C08939=1018.974,60.779,-109.447,166.802,53.022,159.705
C08940=1018.980,61.027,-109.462,166.804,53.016,159.704
C08941=1018.986,61.276,-109.479,166.807,53.009,159.704
C08942=1018.991,61.526,-109.494,166.810,53.001,159.703
C08943=1018.997,61.776,-109.511,166.812,52.995,159.702
C08944=1019.002,62.025,-109.526,166.815,52.987,159.701
C08945=1019.007,62.275,-109.543,166.817,52.981,159.700
C08946=1019.013,62.524,-109.559,166.820,52.973,159.700
C08947=1019.019,62.774,-109.574,166.822,52.967,159.699
C08948=1019.025,63.023,-109.591,166.825,52.960,159.698
C08949=1019.030,63.272,-109.607,166.827,52.953,159.697
C08950=1019.036,63.522,-109.623,166.831,52.946,159.697
C08951=1019.042,63.771,-109.640,166.833,52.939,159.696
C08952=1019.046,64.021,-109.656,166.836,52.932,159.695
C08953=1019.052,64.270,-109.672,166.838,52.926,159.694
C08954=1019.057,64.520,-109.688,166.841,52.918,159.693
C08955=1019.063,64.769,-109.705,166.844,52.912,159.693
C08956=1019.069,65.018,-109.721,166.847,52.905,159.692
C08957=1019.074,65.268,-109.738,166.849,52.898,159.691
C08958=1019.079,65.517,-109.754,166.852,52.891,159.690
C08959=1019.084,65.767,-109.770,166.854,52.884,159.689
C08960=1019.090,66.016,-109.786,166.856,52.878,159.688
C08961=1019.096,66.266,-109.803,166.859,52.871,159.688
C08962=1019.101,66.515,-109.819,166.862,52.865,159.687
C08963=1019.106,66.764,-109.836,166.865,52.857,159.686
C08964=1019.112,67.014,-109.852,166.867,52.851,159.685
C08965=1019.118,67.263,-109.868,166.870,52.843,159.684
C08966=1019.123,67.513,-109.885,166.872,52.837,159.684
C08967=1019.129,67.762,-109.901,166.875,52.830,159.683
C08968=1019.134,68.011,-109.918,166.877,52.823,159.682
C08969=1019.140,68.260,-109.934,166.881,52.816,159.681
C08970=1019.145,68.510,-109.951,166.883,52.810,159.680
C08971=1019.150,68.760,-109.968,166.886,52.802,159.680
C08972=1019.156,69.009,-109.984,166.888,52.796,159.679
C08973=1019.161,69.259,-110.001,166.890,52.789,159.678
C08974=1019.167,69.507,-110.017,166.894,52.782,159.677
C08975=1019.172,69.757,-110.034,166.896,52.776,159.676
C08976=1019.177,70.007,-110.050,166.899,52.769,159.676
C08977=1019.183,70.256,-110.067,166.901,52.762,159.675
C08978=1019.188,70.506,-110.084,166.904,52.755,159.674
C08979=1019.194,70.755,-110.100,166.906,52.748,159.673
C08980=1019.199,71.005,-110.117,166.910,52.742,159.673
C08981=1019.204,71.254,-110.133,166.912,52.735,159.672
C08982=1019.210,71.502,-110.150,166.914,52.728,159.671
C08983=1019.216,71.752,-110.167,166.917,52.721,159.670
C08984=1019.221,72.002,-110.184,166.919,52.714,159.669
C08985=1019.227,72.251,-110.200,166.922,52.707,159.668
C08986=1019.232,72.501,-110.217,166.925,52.701,159.668
C08987=1019.238,72.750,-110.233,166.928,52.694,159.667
C08988=1019.243,73.000,-110.250,166.930,52.687,159.666
C08989=1019.248,73.249,-110.267,166.933,52.680,159.665
C08990=1019.254,73.497,-110.284,166.935,52.673,159.664
C08991=1019.259,73.747,-110.300,166.939,52.666,159.664
C08992=1019.264,73.997,-110.317,166.941,52.659,159.663
C08993=1019.270,74.246,-110.333,166.944,52.653,159.662
C08994=1019.276,74.496,-110.350,166.946,52.646,159.661
C08995=1019.282,74.778,-110.369,166.949,52.638,159.660
C08996=1019.288,75.061,-110.389,166.952,52.631,159.659
C08997=1019.294,75.343,-110.408,166.956,52.622,159.658
C08998=1019.300,75.626,-110.427,166.958,52.615,159.657
C08999=1019.306,75.875,-110.443,166.960,52.608,159.657
C09000=1019.311,76.125,-110.460,166.964,52.601,159.656
C09001=1019.317,76.374,-110.477,166.966,52.595,159.655
C09002=1019.322,76.623,-110.494,166.969,52.588,159.654
C09003=1019.328,76.873,-110.510,166.971,52.581,159.653
C09004=1019.333,77.122,-110.528,166.974,52.574,159.653
C09005=1019.339,77.371,-110.545,166.977,52.567,159.652
C09006=1019.344,77.621,-110.562,166.979,52.560,159.651
C09007=1019.349,77.870,-110.579,166.982,52.554,159.650
C09008=1019.355,78.120,-110.596,166.984,52.547,159.649
C09009=1019.360,78.369,-110.613,166.988,52.540,159.649
C09010=1019.365,78.619,-110.630,166.990,52.533,159.648
C09011=1019.371,78.868,-110.647,166.993,52.527,159.647
C09012=1019.376,79.117,-110.665,166.995,52.520,159.646
C09013=1019.381,79.367,-110.682,166.998,52.514,159.645
C09014=1019.388,79.616,-110.699,167.001,52.506,159.645
C09015=1019.393,79.865,-110.716,167.003,52.500,159.644
C09016=1019.398,80.115,-110.732,167.006,52.493,159.643
C09017=1019.403,80.364,-110.750,167.009,52.487,159.642
C09018=1019.408,80.613,-110.766,167.012,52.480,159.642
C09019=1019.414,80.862,-110.784,167.014,52.473,159.641
C09020=1019.419,81.112,-110.801,167.016,52.466,159.640
C09021=1019.424,81.361,-110.818,167.019,52.459,159.639
C09022=1019.430,81.610,-110.835,167.021,52.452,159.638
C09023=1019.436,81.860,-110.853,167.025,52.446,159.638
C09024=1019.441,82.110,-110.870,167.027,52.439,159.637
C09025=1019.446,82.359,-110.888,167.030,52.432,159.636
C09026=1019.452,82.608,-110.905,167.032,52.425,159.635
C09027=1019.457,82.857,-110.922,167.036,52.418,159.634
C09028=1019.462,83.107,-110.939,167.038,52.412,159.633
C09029=1019.468,83.356,-110.956,167.041,52.404,159.633
C09030=1019.473,83.606,-110.973,167.043,52.398,159.632
C09031=1019.479,83.855,-110.991,167.047,52.391,159.631
C09032=1019.485,84.104,-111.007,167.049,52.385,159.630
C09033=1019.490,84.353,-111.025,167.051,52.378,159.629
C09034=1019.495,84.603,-111.042,167.054,52.371,159.629
C09035=1019.501,84.852,-111.059,167.056,52.364,159.628
C09036=1019.506,85.102,-111.076,167.059,52.357,159.627
C09037=1019.512,85.351,-111.094,167.062,52.350,159.626
C09038=1019.517,85.600,-111.111,167.065,52.343,159.625
C09039=1019.522,85.849,-111.128,167.067,52.337,159.624
C09040=1019.528,86.098,-111.146,167.070,52.330,159.624
C09041=1019.533,86.348,-111.162,167.072,52.323,159.623
C09042=1019.539,86.597,-111.180,167.075,52.316,159.622
C09043=1019.545,86.847,-111.198,167.078,52.309,159.621
C09044=1019.550,87.096,-111.215,167.081,52.302,159.620
C09045=1019.555,87.346,-111.232,167.083,52.295,159.619
C09046=1019.561,87.595,-111.249,167.086,52.288,159.619
C09047=1019.566,87.844,-111.267,167.088,52.282,159.618
C09048=1019.572,88.093,-111.284,167.092,52.275,159.617
C09049=1019.577,88.343,-111.301,167.095,52.267,159.616
C09050=1019.582,88.592,-111.319,167.097,52.261,159.615
C09051=1019.588,88.841,-111.336,167.100,52.254,159.615
C09052=1019.594,89.091,-111.354,167.103,52.248,159.614
C09053=1019.599,89.340,-111.371,167.106,52.241,159.613
C09054=1019.605,89.589,-111.389,167.108,52.234,159.612
C09055=1019.610,89.838,-111.406,167.110,52.227,159.611
C09056=1019.615,90.088,-111.424,167.113,52.220,159.611
C09057=1019.620,90.337,-111.441,167.116,52.214,159.610
C09058=1019.626,90.587,-111.459,167.119,52.207,159.609
C09059=1019.632,90.870,-111.479,167.122,52.199,159.608
C09060=1019.638,91.152,-111.500,167.125,52.192,159.607
C09061=1019.644,91.435,-111.519,167.128,52.184,159.606
C09062=1019.650,91.718,-111.539,167.131,52.177,159.605
C09063=1019.655,91.967,-111.557,167.134,52.170,159.605
C09064=1019.661,92.216,-111.574,167.136,52.163,159.604
C09065=1019.666,92.466,-111.593,167.139,52.156,159.603
C09066=1019.672,92.715,-111.610,167.142,52.150,159.602
C09067=1019.677,92.964,-111.628,167.145,52.142,159.601
C09068=1019.682,93.213,-111.646,167.147,52.136,159.601
C09069=1019.687,93.463,-111.663,167.150,52.129,159.600
C09070=1019.693,93.712,-111.680,167.152,52.122,159.599
C09071=1019.699,93.962,-111.698,167.156,52.116,159.598
C09072=1019.704,94.211,-111.716,167.158,52.109,159.597
C09073=1019.709,94.460,-111.734,167.161,52.102,159.597
C09074=1019.715,94.709,-111.752,167.164,52.095,159.596
C09075=1019.720,94.958,-111.769,167.167,52.088,159.595
C09076=1019.726,95.208,-111.788,167.169,52.082,159.594
C09077=1019.731,95.457,-111.805,167.172,52.075,159.593
C09078=1019.737,95.706,-111.823,167.174,52.068,159.592
C09079=1019.742,95.956,-111.841,167.178,52.061,159.592
C09080=1019.747,96.205,-111.859,167.180,52.054,159.591
C09081=1019.753,96.454,-111.876,167.183,52.047,159.590
C09082=1019.759,96.703,-111.894,167.185,52.041,159.589
C09083=1019.763,96.953,-111.912,167.189,52.034,159.588
C09084=1019.769,97.202,-111.930,167.191,52.027,159.587
C09085=1019.775,97.452,-111.948,167.194,52.020,159.587
C09086=1019.781,97.701,-111.965,167.196,52.013,159.586
C09087=1019.785,97.950,-111.983,167.199,52.006,159.585
C09088=1019.791,98.199,-112.001,167.202,52.000,159.584
C09089=1019.797,98.449,-112.019,167.205,51.993,159.583
C09090=1019.802,98.698,-112.037,167.207,51.986,159.583
C09091=1019.807,98.947,-112.055,167.210,51.979,159.582
C09092=1019.813,99.196,-112.072,167.214,51.972,159.581
C09093=1019.818,99.446,-112.091,167.216,51.965,159.580
C09094=1019.824,99.695,-112.108,167.218,51.959,159.579
C09095=1019.829,99.945,-112.126,167.222,51.952,159.579
C09096=1019.835,100.194,-112.144,167.224,51.946,159.578
C09097=1019.840,100.443,-112.163,167.227,51.939,159.577
C09098=1019.845,100.692,-112.181,167.229,51.932,159.576
C09099=1019.850,100.942,-112.199,167.233,51.925,159.575
C09100=1019.855,101.192,-112.218,167.235,51.918,159.574
C09101=1019.861,101.441,-112.235,167.239,51.912,159.574
C09102=1019.866,101.689,-112.254,167.241,51.905,159.573
C09103=1019.872,101.938,-112.272,167.244,51.898,159.572
C09104=1019.877,102.188,-112.290,167.246,51.892,159.571
C09105=1019.882,102.438,-112.308,167.249,51.885,159.571
C09106=1019.888,102.686,-112.327,167.252,51.878,159.570
C09107=1019.893,102.936,-112.345,167.255,51.871,159.569
C09108=1019.898,103.185,-112.363,167.257,51.864,159.568
C09109=1019.903,103.435,-112.381,167.260,51.857,159.567
C09110=1019.910,103.684,-112.399,167.263,51.851,159.567
C09111=1019.914,103.933,-112.418,167.266,51.844,159.566
C09112=1019.919,104.182,-112.436,167.269,51.838,159.565
C09113=1019.925,104.432,-112.454,167.272,51.831,159.564
C09114=1019.930,104.681,-112.473,167.274,51.824,159.563
C09115=1019.936,104.930,-112.490,167.277,51.817,159.563
C09116=1019.941,105.180,-112.509,167.280,51.811,159.562
C09117=1019.946,105.429,-112.528,167.283,51.804,159.561
C09118=1019.952,105.678,-112.545,167.285,51.797,159.560
C09119=1019.957,105.928,-112.564,167.288,51.790,159.559
C09120=1019.963,106.176,-112.582,167.292,51.783,159.559
C09121=1019.968,106.426,-112.600,167.294,51.776,159.558
C09122=1019.974,106.675,-112.618,167.297,51.769,159.557
C09123=1019.979,106.958,-112.640,167.300,51.762,159.556
C09124=1019.986,107.241,-112.660,167.303,51.754,159.555
C09125=1019.992,107.524,-112.681,167.307,51.746,159.554
C09126=1019.998,107.806,-112.702,167.310,51.738,159.553
C09127=1020.004,108.056,-112.720,167.312,51.732,159.552
C09128=1020.009,108.305,-112.738,167.315,51.725,159.551
C09129=1020.014,108.554,-112.757,167.318,51.718,159.551
C09130=1020.020,108.804,-112.775,167.321,51.711,159.550
C09131=1020.025,109.052,-112.794,167.324,51.704,159.549
C09132=1020.032,109.302,-112.812,167.326,51.698,159.548
C09133=1020.036,109.551,-112.830,167.330,51.691,159.547
C09134=1020.041,109.800,-112.849,167.332,51.684,159.546
C09135=1020.047,110.050,-112.867,167.335,51.678,159.546
C09136=1020.053,110.299,-112.885,167.338,51.671,159.545
C09137=1020.058,110.549,-112.904,167.341,51.664,159.544
C09138=1020.063,110.797,-112.923,167.344,51.657,159.543
C09139=1020.068,111.047,-112.941,167.347,51.651,159.543
C09140=1020.074,111.296,-112.960,167.350,51.644,159.542
C09141=1020.079,111.545,-112.979,167.352,51.637,159.541
C09142=1020.085,111.795,-112.997,167.355,51.630,159.540
C09143=1020.090,112.043,-113.016,167.358,51.623,159.539
C09144=1020.095,112.293,-113.034,167.361,51.616,159.539
C09145=1020.100,112.542,-113.053,167.363,51.610,159.538
C09146=1020.106,112.792,-113.073,167.367,51.603,159.537
C09147=1020.111,113.041,-113.091,167.369,51.597,159.536
C09148=1020.116,113.290,-113.110,167.373,51.590,159.535
C09149=1020.122,113.539,-113.129,167.375,51.583,159.535
C09150=1020.127,113.789,-113.147,167.378,51.576,159.534
C09151=1020.132,114.038,-113.166,167.380,51.570,159.533
C09152=1020.137,114.287,-113.185,167.384,51.564,159.532
C09153=1020.143,114.536,-113.204,167.386,51.557,159.531
C09154=1020.148,114.785,-113.223,167.390,51.550,159.531
C09155=1020.153,115.035,-113.242,167.392,51.543,159.530
C09156=1020.158,115.284,-113.261,167.395,51.536,159.529
C09157=1020.164,115.533,-113.280,167.398,51.530,159.528
C09158=1020.169,115.782,-113.298,167.401,51.523,159.527
C09159=1020.175,116.032,-113.317,167.404,51.517,159.527
C09160=1020.179,116.281,-113.337,167.407,51.510,159.526
C09161=1020.185,116.530,-113.356,167.409,51.504,159.525
C09162=1020.190,116.779,-113.375,167.412,51.497,159.524
C09163=1020.195,117.029,-113.393,167.415,51.490,159.523
C09164=1020.200,117.278,-113.412,167.418,51.483,159.523
C09165=1020.206,117.527,-113.432,167.421,51.476,159.522
C09166=1020.211,117.776,-113.450,167.424,51.470,159.521
C09167=1020.217,118.025,-113.470,167.427,51.463,159.520
C09168=1020.222,118.274,-113.489,167.430,51.457,159.520
C09169=1020.227,118.524,-113.507,167.433,51.450,159.519
C09170=1020.232,118.773,-113.526,167.435,51.443,159.518
C09171=1020.238,119.022,-113.545,167.439,51.436,159.517
C09172=1020.243,119.271,-113.564,167.441,51.430,159.516
C09173=1020.249,119.521,-113.583,167.444,51.423,159.516
C09174=1020.254,119.770,-113.603,167.448,51.416,159.515
C09175=1020.259,120.019,-113.622,167.450,51.409,159.514
C09176=1020.264,120.268,-113.641,167.454,51.403,159.513
C09177=1020.269,120.517,-113.660,167.456,51.396,159.512
C09178=1020.275,120.767,-113.679,167.459,51.390,159.512
C09179=1020.280,121.016,-113.698,167.463,51.383,159.511
C09180=1020.286,121.265,-113.717,167.465,51.376,159.510
C09181=1020.291,121.515,-113.736,167.468,51.369,159.509
C09182=1020.296,121.764,-113.755,167.471,51.363,159.508
C09183=1020.302,122.013,-113.774,167.474,51.356,159.508
C09184=1020.307,122.262,-113.793,167.477,51.349,159.507
C09185=1020.313,122.511,-113.812,167.480,51.342,159.506
C09186=1020.318,122.761,-113.832,167.483,51.335,159.505
C09187=1020.324,123.043,-113.853,167.486,51.328,159.504
C09188=1020.330,123.326,-113.875,167.490,51.320,159.503
C09189=1020.336,123.609,-113.897,167.493,51.312,159.502
C09190=1020.342,123.891,-113.918,167.496,51.305,159.502
C09191=1020.348,124.141,-113.938,167.499,51.298,159.501
C09192=1020.353,124.389,-113.957,167.503,51.291,159.500
C09193=1020.359,124.639,-113.976,167.505,51.285,159.499
C09194=1020.364,124.889,-113.996,167.508,51.278,159.498
C09195=1020.369,125.137,-114.015,167.512,51.271,159.498
C09196=1020.375,125.387,-114.034,167.514,51.264,159.497
C09197=1020.380,125.636,-114.053,167.517,51.257,159.496
C09198=1020.385,125.885,-114.072,167.520,51.251,159.495
C09199=1020.391,126.134,-114.091,167.523,51.244,159.494
C09200=1020.397,126.384,-114.110,167.526,51.237,159.494
C09201=1020.402,126.633,-114.129,167.530,51.230,159.493
C09202=1020.408,126.882,-114.148,167.532,51.224,159.492
C09203=1020.413,127.131,-114.168,167.536,51.217,159.491
C09204=1020.418,127.380,-114.188,167.539,51.210,159.490
C09205=1020.424,127.629,-114.207,167.541,51.203,159.489
C09206=1020.429,127.879,-114.226,167.544,51.196,159.489
C09207=1020.435,128.128,-114.246,167.548,51.189,159.488
C09208=1020.440,128.377,-114.265,167.550,51.182,159.487
C09209=1020.446,128.626,-114.284,167.553,51.175,159.486
C09210=1020.451,128.876,-114.303,167.557,51.169,159.485
C09211=1020.456,129.124,-114.322,167.559,51.162,159.484
C09212=1020.462,129.374,-114.341,167.562,51.155,159.484
C09213=1020.468,129.623,-114.361,167.566,51.148,159.483
C09214=1020.473,129.872,-114.381,167.569,51.141,159.482
C09215=1020.478,130.121,-114.400,167.571,51.135,159.481
C09216=1020.484,130.371,-114.419,167.575,51.128,159.481
C09217=1020.489,130.620,-114.440,167.577,51.122,159.480
C09218=1020.495,130.869,-114.459,167.581,51.115,159.479
C09219=1020.500,131.119,-114.479,167.584,51.108,159.478
C09220=1020.505,131.368,-114.498,167.587,51.102,159.477
C09221=1020.510,131.617,-114.518,167.590,51.095,159.477
C09222=1020.516,131.866,-114.537,167.593,51.088,159.476
C09223=1020.520,132.115,-114.558,167.596,51.082,159.475
C09224=1020.526,132.364,-114.577,167.599,51.075,159.474
C09225=1020.532,132.614,-114.596,167.603,51.068,159.474
C09226=1020.537,132.863,-114.617,167.605,51.062,159.473
C09227=1020.543,133.112,-114.636,167.609,51.055,159.472
C09228=1020.547,133.361,-114.655,167.611,51.049,159.471
C09229=1020.553,133.610,-114.675,167.614,51.042,159.470
C09230=1020.558,133.860,-114.695,167.618,51.035,159.470
C09231=1020.564,134.108,-114.715,167.620,51.028,159.469
C09232=1020.568,134.358,-114.735,167.623,51.021,159.468
C09233=1020.574,134.606,-114.754,167.627,51.015,159.467
C09234=1020.579,134.856,-114.774,167.630,51.008,159.466
C09235=1020.585,135.106,-114.794,167.633,51.001,159.466
C09236=1020.591,135.354,-114.814,167.636,50.995,159.465
C09237=1020.595,135.603,-114.833,167.640,50.988,159.464
C09238=1020.601,135.852,-114.853,167.642,50.982,159.463
C09239=1020.606,136.102,-114.873,167.645,50.975,159.463
C09240=1020.612,136.351,-114.893,167.649,50.968,159.462
C09241=1020.617,136.600,-114.913,167.651,50.961,159.461
C09242=1020.623,136.850,-114.933,167.655,50.955,159.460
C09243=1020.628,137.098,-114.952,167.658,50.948,159.459
C09244=1020.633,137.347,-114.973,167.660,50.941,159.459
C09245=1020.639,137.596,-114.993,167.664,50.934,159.458
C09246=1020.644,137.846,-115.012,167.668,50.928,159.457
C09247=1020.650,138.095,-115.032,167.671,50.921,159.456
C09248=1020.655,138.345,-115.052,167.673,50.915,159.456
C09249=1020.659,138.593,-115.072,167.677,50.908,159.455
C09250=1020.665,138.842,-115.092,167.680,50.901,159.454
C09251=1020.671,139.125,-115.115,167.683,50.894,159.453
C09252=1020.677,139.408,-115.138,167.687,50.887,159.452
C09253=1020.684,139.690,-115.161,167.691,50.879,159.451
C09254=1020.689,139.973,-115.184,167.694,50.871,159.450
C09255=1020.695,140.222,-115.204,167.697,50.864,159.450
C09256=1020.700,140.472,-115.224,167.701,50.858,159.449
C09257=1020.705,140.720,-115.244,167.703,50.852,159.448
C09258=1020.710,140.969,-115.264,167.707,50.845,159.447
C09259=1020.716,141.219,-115.284,167.710,50.838,159.447
C09260=1020.721,141.468,-115.304,167.712,50.832,159.446
C09261=1020.726,141.717,-115.325,167.716,50.825,159.445
C09262=1020.732,141.966,-115.345,167.719,50.818,159.444
C09263=1020.737,142.215,-115.365,167.723,50.812,159.444
C09264=1020.743,142.464,-115.385,167.725,50.805,159.443
C09265=1020.748,142.714,-115.406,167.729,50.799,159.442
C09266=1020.754,142.962,-115.426,167.732,50.792,159.441
C09267=1020.759,143.212,-115.445,167.735,50.785,159.440
C09268=1020.763,143.461,-115.466,167.738,50.778,159.440
C09269=1020.769,143.710,-115.486,167.742,50.772,159.439
C09270=1020.775,143.959,-115.506,167.745,50.765,159.438
C09271=1020.780,144.208,-115.527,167.748,50.759,159.437
C09272=1020.785,144.457,-115.547,167.751,50.752,159.437
C09273=1020.790,144.707,-115.567,167.755,50.745,159.436
C09274=1020.796,144.955,-115.587,167.758,50.738,159.435
C09275=1020.801,145.204,-115.608,167.760,50.732,159.434
C09276=1020.807,145.454,-115.628,167.764,50.725,159.433
C09277=1020.813,145.702,-115.648,167.767,50.718,159.433
C09278=1020.818,145.952,-115.669,167.771,50.712,159.432
C09279=1020.823,146.201,-115.689,167.774,50.706,159.431
C09280=1020.828,146.450,-115.710,167.777,50.699,159.430
C09281=1020.834,146.699,-115.730,167.780,50.692,159.430
C09282=1020.839,146.949,-115.750,167.784,50.685,159.429
C09283=1020.844,147.198,-115.771,167.787,50.680,159.428
C09284=1020.849,147.447,-115.791,167.790,50.673,159.427
C09285=1020.854,147.696,-115.812,167.794,50.666,159.427
C09286=1020.860,147.945,-115.832,167.797,50.659,159.426
C09287=1020.865,148.194,-115.854,167.800,50.653,159.425
C09288=1020.870,148.443,-115.874,167.803,50.647,159.424
C09289=1020.876,148.692,-115.895,167.807,50.640,159.424
C09290=1020.881,148.941,-115.915,167.810,50.633,159.423
C09291=1020.886,149.190,-115.936,167.812,50.626,159.422
C09292=1020.891,149.439,-115.956,167.816,50.620,159.421
C09293=1020.897,149.688,-115.977,167.820,50.614,159.421
C09294=1020.902,149.938,-115.998,167.823,50.607,159.420
C09295=1020.907,150.187,-116.018,167.826,50.600,159.419
C09296=1020.912,150.436,-116.039,167.829,50.594,159.418
C09297=1020.918,150.685,-116.059,167.833,50.587,159.418
C09298=1020.923,150.934,-116.080,167.836,50.581,159.417
C09299=1020.929,151.183,-116.101,167.839,50.574,159.416
C09300=1020.934,151.432,-116.122,167.842,50.567,159.415
C09301=1020.940,151.681,-116.142,167.846,50.561,159.415
C09302=1020.945,151.931,-116.163,167.850,50.554,159.414
C09303=1020.950,152.180,-116.184,167.853,50.548,159.413
C09304=1020.955,152.429,-116.204,167.855,50.541,159.412
C09305=1020.961,152.677,-116.225,167.859,50.534,159.411
C09306=1020.966,152.926,-116.246,167.863,50.528,159.411
C09307=1020.971,153.176,-116.267,167.866,50.522,159.410
C09308=1020.977,153.425,-116.287,167.870,50.515,159.409
C09309=1020.982,153.674,-116.308,167.872,50.508,159.408
C09310=1020.988,153.923,-116.329,167.876,50.502,159.408
C09311=1020.993,154.172,-116.350,167.879,50.495,159.407
C09312=1020.999,154.421,-116.370,167.883,50.489,159.406
C09313=1021.003,154.670,-116.392,167.887,50.483,159.406
C09314=1021.009,154.919,-116.413,167.889,50.476,159.405
C09315=1021.015,155.201,-116.437,167.893,50.468,159.404
C09316=1021.021,155.484,-116.460,167.897,50.462,159.403
C09317=1021.027,155.766,-116.484,167.901,50.454,159.402
C09318=1021.033,156.050,-116.507,167.905,50.446,159.402
C09319=1021.039,156.298,-116.529,167.908,50.440,159.401
C09320=1021.043,156.548,-116.550,167.911,50.433,159.400
C09321=1021.049,156.797,-116.570,167.915,50.427,159.399
C09322=1021.054,157.045,-116.592,167.918,50.420,159.399
C09323=1021.059,157.294,-116.612,167.922,50.414,159.398
C09324=1021.066,157.543,-116.634,167.926,50.407,159.397
C09325=1021.071,157.793,-116.654,167.928,50.401,159.396
C09326=1021.075,158.042,-116.676,167.931,50.394,159.396
C09327=1021.081,158.291,-116.697,167.935,50.388,159.395
C09328=1021.086,158.540,-116.717,167.939,50.381,159.394
C09329=1021.092,158.789,-116.739,167.942,50.374,159.393
C09330=1021.098,159.038,-116.760,167.946,50.368,159.393
C09331=1021.102,159.287,-116.781,167.949,50.362,159.392
C09332=1021.107,159.536,-116.803,167.952,50.356,159.391
C09333=1021.113,159.785,-116.824,167.956,50.349,159.391
C09334=1021.117,160.034,-116.846,167.959,50.342,159.390
C09335=1021.123,160.283,-116.868,167.962,50.337,159.389
C09336=1021.128,160.532,-116.888,167.966,50.330,159.388
C09337=1021.133,160.781,-116.910,167.970,50.324,159.388
C09338=1021.138,161.030,-116.932,167.973,50.317,159.387
C09339=1021.143,161.279,-116.953,167.976,50.311,159.386
C09340=1021.148,161.528,-116.975,167.979,50.304,159.386
C09341=1021.154,161.777,-116.996,167.983,50.298,159.385
C09342=1021.159,162.026,-117.018,167.987,50.292,159.384
C09343=1021.163,162.275,-117.039,167.991,50.286,159.384
C09344=1021.169,162.524,-117.061,167.993,50.279,159.383
C09345=1021.174,162.773,-117.083,167.997,50.273,159.382
C09346=1021.180,163.022,-117.104,168.000,50.266,159.381
C09347=1021.184,163.271,-117.125,168.004,50.260,159.381
C09348=1021.189,163.520,-117.147,168.008,50.254,159.380
C09349=1021.195,163.769,-117.169,168.011,50.248,159.379
C09350=1021.200,164.018,-117.191,168.014,50.241,159.379
C09351=1021.205,164.267,-117.212,168.018,50.235,159.378
C09352=1021.211,164.517,-117.233,168.022,50.228,159.377
C09353=1021.216,164.765,-117.255,168.025,50.222,159.377
C09354=1021.221,165.014,-117.277,168.028,50.216,159.376
C09355=1021.226,165.263,-117.298,168.031,50.209,159.375
C09356=1021.231,165.512,-117.321,168.035,50.203,159.374
C09357=1021.237,165.761,-117.342,168.039,50.196,159.374
C09358=1021.242,166.010,-117.363,168.043,50.190,159.373
C09359=1021.247,166.260,-117.385,168.046,50.184,159.372
C09360=1021.253,166.508,-117.406,168.050,50.178,159.372
C09361=1021.257,166.757,-117.428,168.053,50.171,159.371
C09362=1021.263,167.007,-117.451,168.056,50.165,159.370
C09363=1021.268,167.255,-117.472,168.060,50.158,159.370
C09364=1021.273,167.504,-117.494,168.064,50.152,159.369
C09365=1021.279,167.753,-117.516,168.067,50.146,159.368
C09366=1021.284,168.002,-117.537,168.071,50.140,159.368
C09367=1021.289,168.251,-117.559,168.075,50.133,159.367
C09368=1021.294,168.500,-117.581,168.078,50.126,159.366
C09369=1021.300,168.749,-117.603,168.082,50.120,159.365
C09370=1021.305,168.998,-117.624,168.085,50.114,159.365
C09371=1021.311,169.247,-117.645,168.089,50.108,159.364
C09372=1021.315,169.496,-117.667,168.092,50.101,159.363
C09373=1021.321,169.746,-117.689,168.096,50.095,159.363
C09374=1021.326,169.994,-117.711,168.100,50.088,159.362
C09375=1021.331,170.243,-117.733,168.103,50.082,159.361
C09376=1021.337,170.493,-117.755,168.107,50.076,159.360
C09377=1021.342,170.741,-117.776,168.111,50.070,159.360
C09378=1021.348,170.990,-117.799,168.114,50.063,159.359
C09379=1021.354,171.272,-117.823,168.119,50.056,159.358
C09380=1021.360,171.554,-117.849,168.122,50.048,159.357
C09381=1021.366,171.836,-117.873,168.127,50.041,159.357
C09382=1021.372,172.118,-117.898,168.131,50.034,159.356
C09383=1021.377,172.367,-117.920,168.135,50.028,159.355
C09384=1021.383,172.617,-117.942,168.138,50.021,159.355
C09385=1021.388,172.865,-117.963,168.142,50.015,159.354
C09386=1021.394,173.115,-117.985,168.146,50.008,159.353
C09387=1021.398,173.364,-118.007,168.150,50.002,159.353
C09388=1021.405,173.613,-118.029,168.153,49.996,159.352
C09389=1021.409,173.862,-118.051,168.157,49.989,159.351
C09390=1021.415,174.111,-118.074,168.161,49.983,159.350
C09391=1021.421,174.359,-118.095,168.164,49.976,159.350
C09392=1021.426,174.609,-118.117,168.168,49.970,159.349
C09393=1021.431,174.857,-118.139,168.171,49.964,159.348
C09394=1021.437,175.107,-118.161,168.175,49.957,159.348
C09395=1021.442,175.355,-118.183,168.179,49.951,159.347
C09396=1021.448,175.604,-118.205,168.183,49.945,159.346
C09397=1021.453,175.853,-118.227,168.186,49.938,159.346
C09398=1021.459,176.102,-118.249,168.190,49.931,159.345
C09399=1021.464,176.352,-118.271,168.194,49.925,159.344
C09400=1021.470,176.600,-118.293,168.197,49.919,159.343
C09401=1021.475,176.849,-118.315,168.201,49.913,159.343
C09402=1021.480,177.098,-118.337,168.205,49.906,159.342
C09403=1021.486,177.347,-118.359,168.209,49.900,159.341
C09404=1021.492,177.595,-118.381,168.212,49.893,159.341
C09405=1021.497,177.845,-118.404,168.216,49.887,159.340
C09406=1021.502,178.095,-118.426,168.220,49.881,159.339
C09407=1021.508,178.343,-118.447,168.223,49.874,159.339
C09408=1021.514,178.592,-118.470,168.227,49.868,159.338
C09409=1021.518,178.841,-118.492,168.231,49.861,159.337
C09410=1021.525,179.090,-118.514,168.236,49.855,159.337
C09411=1021.530,179.339,-118.537,168.239,49.848,159.336
C09412=1021.535,179.588,-118.558,168.243,49.842,159.335
C09413=1021.541,179.837,-118.580,168.247,49.836,159.335
C09414=1021.547,180.086,-118.603,168.251,49.830,159.334
C09415=1021.552,180.335,-118.625,168.254,49.823,159.333
C09416=1021.558,180.584,-118.647,168.258,49.817,159.333
C09417=1021.564,180.833,-118.669,168.262,49.810,159.332
C09418=1021.569,181.081,-118.691,168.265,49.804,159.331
C09419=1021.575,181.330,-118.714,168.270,49.798,159.331
C09420=1021.581,181.580,-118.736,168.274,49.791,159.330
C09421=1021.586,181.828,-118.759,168.278,49.785,159.329
C09422=1021.591,182.077,-118.781,168.281,49.778,159.328
C09423=1021.597,182.327,-118.803,168.285,49.772,159.328
C09424=1021.602,182.575,-118.826,168.289,49.766,159.327
C09425=1021.607,182.824,-118.848,168.293,49.760,159.326
C09426=1021.612,183.074,-118.871,168.297,49.754,159.326
C09427=1021.618,183.323,-118.894,168.301,49.748,159.325
C09428=1021.623,183.571,-118.917,168.305,49.742,159.325
C09429=1021.628,183.820,-118.940,168.308,49.736,159.324
C09430=1021.633,184.070,-118.963,168.312,49.729,159.323
C09431=1021.638,184.318,-118.985,168.316,49.723,159.323
C09432=1021.644,184.567,-119.008,168.320,49.717,159.322
C09433=1021.649,184.816,-119.032,168.324,49.711,159.322
C09434=1021.654,185.064,-119.054,168.327,49.705,159.321
C09435=1021.660,185.314,-119.076,168.331,49.699,159.320
C09436=1021.665,185.563,-119.100,168.335,49.693,159.320
C09437=1021.670,185.811,-119.123,168.339,49.687,159.319
C09438=1021.676,186.060,-119.146,168.343,49.681,159.318
C09439=1021.681,186.309,-119.169,168.347,49.674,159.318
C09440=1021.686,186.558,-119.192,168.351,49.668,159.317
C09441=1021.691,186.806,-119.215,168.355,49.662,159.316
C09442=1021.696,187.056,-119.237,168.359,49.656,159.316
C09443=1021.702,187.338,-119.264,168.363,49.649,159.315
C09444=1021.708,187.619,-119.290,168.368,49.642,159.314
C09445=1021.714,187.901,-119.316,168.372,49.635,159.314
C09446=1021.720,188.183,-119.342,168.377,49.628,159.313
C09447=1021.726,188.431,-119.364,168.381,49.622,159.312
C09448=1021.731,188.680,-119.387,168.385,49.616,159.312
C09449=1021.736,188.929,-119.411,168.388,49.610,159.311
C09450=1021.742,189.178,-119.434,168.392,49.604,159.310
C09451=1021.748,189.427,-119.457,168.396,49.598,159.310
C09452=1021.752,189.676,-119.480,168.401,49.591,159.309
C09453=1021.758,189.924,-119.503,168.405,49.585,159.309
C09454=1021.764,190.173,-119.526,168.409,49.579,159.308
C09455=1021.769,190.423,-119.549,168.413,49.573,159.307
C09456=1021.774,190.671,-119.572,168.417,49.567,159.307
C09457=1021.780,190.920,-119.595,168.420,49.561,159.306
C09458=1021.784,191.169,-119.619,168.424,49.555,159.305
C09459=1021.790,191.418,-119.641,168.429,49.549,159.305
C09460=1021.796,191.667,-119.664,168.433,49.543,159.304
C09461=1021.801,191.916,-119.688,168.437,49.537,159.304
C09462=1021.807,192.165,-119.711,168.441,49.531,159.303
C09463=1021.813,192.413,-119.735,168.445,49.524,159.302
C09464=1021.818,192.662,-119.758,168.449,49.518,159.302
C09465=1021.823,192.911,-119.781,168.454,49.512,159.301
C09466=1021.828,193.160,-119.804,168.458,49.506,159.301
C09467=1021.834,193.409,-119.827,168.462,49.500,159.300
C09468=1021.839,193.657,-119.850,168.465,49.493,159.299
C09469=1021.844,193.907,-119.874,168.469,49.488,159.299
C09470=1021.850,194.156,-119.897,168.474,49.481,159.298
C09471=1021.856,194.404,-119.920,168.478,49.475,159.298
C09472=1021.861,194.653,-119.944,168.482,49.469,159.297
C09473=1021.867,194.902,-119.967,168.486,49.464,159.296
C09474=1021.872,195.151,-119.990,168.490,49.457,159.296
C09475=1021.877,195.400,-120.013,168.495,49.451,159.295
C09476=1021.883,195.648,-120.037,168.499,49.445,159.295
C09477=1021.889,195.897,-120.060,168.503,49.439,159.294
C09478=1021.894,196.146,-120.083,168.507,49.433,159.293
C09479=1021.900,196.395,-120.106,168.512,49.427,159.293
C09480=1021.905,196.644,-120.131,168.516,49.421,159.292
C09481=1021.911,196.893,-120.154,168.519,49.414,159.291
C09482=1021.917,197.142,-120.176,168.523,49.408,159.291
C09483=1021.922,197.390,-120.201,168.528,49.402,159.290
C09484=1021.928,197.639,-120.224,168.532,49.396,159.290
C09485=1021.933,197.888,-120.247,168.536,49.390,159.289
C09486=1021.939,198.137,-120.271,168.540,49.384,159.289
C09487=1021.944,198.386,-120.294,168.545,49.378,159.288
C09488=1021.950,198.634,-120.317,168.549,49.372,159.287
C09489=1021.956,198.883,-120.341,168.553,49.366,159.287
C09490=1021.961,199.132,-120.364,168.558,49.359,159.286
C09491=1021.966,199.381,-120.387,168.562,49.354,159.286
C09492=1021.972,199.629,-120.411,168.566,49.348,159.285
C09493=1021.977,199.879,-120.435,168.571,49.341,159.284
C09494=1021.984,200.128,-120.459,168.575,49.336,159.284
C09495=1021.989,200.377,-120.482,168.579,49.330,159.283
C09496=1021.994,200.625,-120.507,168.583,49.324,159.283
C09497=1021.999,200.874,-120.531,168.586,49.318,159.282
C09498=1022.005,201.123,-120.554,168.591,49.312,159.281
C09499=1022.011,201.371,-120.578,168.595,49.306,159.281
C09500=1022.016,201.621,-120.602,168.599,49.300,159.280
C09501=1022.021,201.869,-120.626,168.604,49.294,159.280
C09502=1022.027,202.118,-120.649,168.608,49.288,159.279
C09503=1022.032,202.367,-120.673,168.613,49.283,159.279
C09504=1022.037,202.615,-120.697,168.617,49.277,159.278
C09505=1022.043,202.865,-120.722,168.622,49.270,159.278
C09506=1022.049,203.114,-120.745,168.626,49.265,159.277
C09507=1022.077,204.361,-120.866,169.059,49.356,159.363
C09508=1022.082,204.574,-120.889,169.061,49.352,159.363
C09509=1022.088,204.787,-120.910,169.065,49.348,159.363
C09510=1022.093,205.000,-120.932,169.067,49.343,159.362
C09511=1022.099,205.213,-120.954,169.071,49.339,159.362
C09512=1022.104,205.425,-120.975,169.073,49.334,159.361
C09513=1022.109,205.639,-120.998,169.077,49.330,159.361
C09514=1022.115,205.852,-121.019,169.079,49.326,159.360
C09515=1022.121,206.100,-121.045,169.083,49.321,159.360
C09516=1022.128,206.349,-121.071,169.086,49.317,159.359
C09517=1022.134,206.598,-121.096,169.089,49.312,159.359
C09518=1022.141,206.846,-121.122,169.093,49.307,159.358
C09519=1022.147,207.095,-121.147,169.096,49.302,159.358
C09520=1022.153,207.343,-121.173,169.100,49.297,159.357
C09521=1022.159,207.592,-121.198,169.103,49.292,159.357
C09522=1022.166,207.840,-121.224,169.107,49.287,159.356
C09523=1022.171,208.089,-121.250,169.110,49.282,159.356
C09524=1022.178,208.339,-121.276,169.113,49.277,159.355
C09525=1022.185,208.587,-121.302,169.117,49.272,159.355
C09526=1022.191,208.835,-121.327,169.120,49.267,159.354
C09527=1022.197,209.083,-121.353,169.123,49.262,159.353
C09528=1022.203,209.332,-121.379,169.127,49.258,159.353
C09529=1022.210,209.581,-121.404,169.130,49.253,159.352
C09530=1022.216,209.830,-121.431,169.134,49.248,159.352
C09531=1022.222,210.078,-121.456,169.138,49.243,159.352
C09532=1022.229,210.326,-121.482,169.141,49.238,159.351
C09533=1022.235,210.575,-121.508,169.144,49.234,159.351
C09534=1022.241,210.823,-121.534,169.148,49.229,159.350
C09535=1022.247,211.072,-121.560,169.151,49.224,159.349
C09536=1022.254,211.321,-121.586,169.155,49.220,159.349
C09537=1022.260,211.570,-121.612,169.158,49.215,159.349
C09538=1022.266,211.818,-121.638,169.161,49.210,159.348
C09539=1022.272,212.067,-121.663,169.164,49.205,159.348
C09540=1022.278,212.315,-121.690,169.168,49.201,159.347
C09541=1022.285,212.564,-121.716,169.171,49.196,159.347
C09542=1022.291,212.812,-121.742,169.175,49.191,159.346
C09543=1022.297,213.061,-121.768,169.178,49.187,159.346
C09544=1022.303,213.309,-121.794,169.182,49.182,159.345
C09545=1022.310,213.558,-121.820,169.185,49.177,159.345
C09546=1022.316,213.807,-121.846,169.190,49.172,159.344
C09547=1022.322,214.055,-121.872,169.193,49.168,159.344
C09548=1022.329,214.303,-121.898,169.196,49.163,159.343
C09549=1022.335,214.553,-121.924,169.200,49.158,159.343
C09550=1022.342,214.801,-121.951,169.203,49.154,159.343
C09551=1022.348,215.049,-121.977,169.206,49.149,159.342
C09552=1022.354,215.299,-122.003,169.210,49.145,159.342
C09553=1022.361,215.547,-122.029,169.213,49.140,159.341
C09554=1022.367,215.795,-122.055,169.217,49.135,159.341
C09555=1022.373,216.044,-122.081,169.220,49.131,159.340
C09556=1022.380,216.292,-122.107,169.224,49.126,159.340
C09557=1022.386,216.541,-122.133,169.227,49.121,159.339
C09558=1022.392,216.789,-122.160,169.231,49.117,159.339
C09559=1022.399,217.038,-122.186,169.234,49.112,159.338
C09560=1022.405,217.287,-122.212,169.238,49.108,159.338
C09561=1022.411,217.535,-122.238,169.241,49.103,159.337
C09562=1022.418,217.783,-122.265,169.245,49.098,159.337
C09563=1022.424,218.032,-122.291,169.249,49.093,159.337
C09564=1022.430,218.280,-122.317,169.252,49.089,159.336
C09565=1022.437,218.529,-122.343,169.256,49.084,159.336
C09566=1022.443,218.778,-122.370,169.259,49.080,159.335
C09567=1022.449,218.993,-122.393,169.262,49.076,159.335
C09568=1022.454,219.207,-122.415,169.265,49.072,159.334
C09569=1022.460,219.422,-122.439,169.269,49.068,159.334
C09570=1022.464,219.637,-122.462,169.271,49.064,159.334
C09571=1022.470,219.852,-122.484,169.274,49.060,159.333
C09572=1022.475,220.067,-122.507,169.278,49.057,159.333
C09573=1022.481,220.281,-122.530,169.280,49.053,159.333
C09574=1022.486,220.496,-122.553,169.283,49.049,159.332
C09575=1022.493,220.745,-122.580,169.287,49.045,159.332
C09576=1022.499,220.993,-122.606,169.290,49.040,159.331
C09577=1022.505,221.241,-122.633,169.294,49.036,159.331
C09578=1022.512,221.490,-122.659,169.297,49.032,159.331
C09579=1022.517,221.739,-122.686,169.301,49.027,159.330
C09580=1022.525,221.987,-122.712,169.304,49.023,159.330
C09581=1022.530,222.236,-122.739,169.308,49.018,159.329
C09582=1022.536,222.484,-122.766,169.311,49.014,159.329
C09583=1022.543,222.733,-122.792,169.315,49.009,159.329
C09584=1022.549,222.981,-122.819,169.319,49.005,159.328
C09585=1022.555,223.230,-122.846,169.322,49.000,159.328
C09586=1022.562,223.478,-122.872,169.326,48.996,159.327
C09587=1022.568,223.727,-122.899,169.329,48.992,159.327
C09588=1022.574,223.975,-122.926,169.333,48.988,159.327
C09589=1022.581,224.224,-122.953,169.336,48.983,159.326
C09590=1022.587,224.472,-122.979,169.340,48.979,159.326
C09591=1022.593,224.721,-123.006,169.344,48.975,159.325
C09592=1022.600,224.969,-123.032,169.347,48.970,159.325
C09593=1022.606,225.218,-123.059,169.351,48.966,159.324
C09594=1022.612,225.467,-123.086,169.354,48.961,159.324
C09595=1022.619,225.714,-123.113,169.358,48.957,159.324
C09596=1022.625,225.963,-123.140,169.362,48.953,159.323
C09597=1022.631,226.212,-123.166,169.366,48.949,159.323
C09598=1022.638,226.460,-123.193,169.370,48.944,159.323
C09599=1022.644,226.709,-123.220,169.373,48.940,159.322
C09600=1022.652,226.957,-123.247,169.377,48.935,159.322
C09601=1022.657,227.205,-123.273,169.381,48.931,159.322
C09602=1022.664,227.454,-123.300,169.383,48.927,159.321
C09603=1022.670,227.702,-123.328,169.387,48.923,159.321
C09604=1022.676,227.951,-123.355,169.391,48.919,159.320
C09605=1022.682,228.199,-123.381,169.394,48.915,159.320
C09606=1022.689,228.448,-123.409,169.398,48.911,159.320
C09607=1022.695,228.697,-123.436,169.402,48.907,159.319
C09608=1022.701,228.945,-123.463,169.405,48.902,159.319
C09609=1022.707,229.194,-123.490,169.409,48.898,159.319
C09610=1022.714,229.442,-123.517,169.413,48.894,159.318
C09611=1022.721,229.690,-123.544,169.416,48.890,159.318
C09612=1022.726,229.939,-123.571,169.420,48.886,159.318
C09613=1022.733,230.188,-123.598,169.424,48.882,159.317
C09614=1022.739,230.435,-123.625,169.427,48.877,159.317
C09615=1022.745,230.684,-123.652,169.431,48.873,159.317
C09616=1022.752,230.933,-123.680,169.435,48.869,159.316
C09617=1022.758,231.181,-123.707,169.438,48.865,159.316
C09618=1022.764,231.430,-123.734,169.442,48.861,159.315
C09619=1022.770,231.677,-123.762,169.446,48.857,159.315
C09620=1022.777,231.926,-123.789,169.449,48.852,159.315
C09621=1022.783,232.175,-123.817,169.453,48.849,159.315
C09622=1022.789,232.423,-123.843,169.457,48.845,159.314
C09623=1022.795,232.672,-123.872,169.461,48.841,159.314
C09624=1022.801,232.920,-123.898,169.465,48.836,159.314
C09625=1022.808,233.169,-123.926,169.468,48.832,159.313
C09626=1022.814,233.417,-123.954,169.471,48.828,159.313
C09627=1022.824,233.793,-123.994,169.477,48.823,159.312
C09628=1022.834,234.169,-124.036,169.482,48.817,159.312
C09629=1022.843,234.546,-124.077,169.488,48.810,159.311
C09630=1022.853,234.922,-124.119,169.494,48.805,159.311
C09631=1022.859,235.170,-124.146,169.497,48.801,159.311
C09632=1022.865,235.419,-124.174,169.501,48.796,159.310
C09633=1022.872,235.667,-124.201,169.505,48.792,159.310
C09634=1022.878,235.915,-124.229,169.509,48.789,159.310
C09635=1022.884,236.165,-124.256,169.512,48.785,159.309
C09636=1022.891,236.413,-124.284,169.516,48.780,159.309
C09637=1022.897,236.661,-124.311,169.520,48.776,159.309
C09638=1022.903,236.909,-124.339,169.524,48.773,159.309
C09639=1022.910,237.158,-124.367,169.527,48.769,159.308
C09640=1022.916,237.407,-124.394,169.531,48.765,159.308
C09641=1022.922,237.654,-124.421,169.535,48.761,159.308
C09642=1022.929,237.903,-124.449,169.539,48.757,159.307
C09643=1022.935,238.152,-124.477,169.543,48.753,159.307
C09644=1022.942,238.400,-124.505,169.547,48.749,159.307
C09645=1022.948,238.648,-124.532,169.550,48.745,159.306
C09646=1022.954,238.897,-124.559,169.554,48.741,159.306
C09647=1022.961,239.145,-124.587,169.558,48.737,159.306
C09648=1022.968,239.394,-124.615,169.562,48.733,159.306
C09649=1022.973,239.642,-124.643,169.566,48.730,159.305
C09650=1022.980,239.890,-124.670,169.569,48.726,159.305
C09651=1022.986,240.139,-124.698,169.572,48.722,159.305
C09652=1022.992,240.387,-124.727,169.576,48.718,159.304
C09653=1022.998,240.635,-124.754,169.580,48.715,159.304
C09654=1023.004,240.884,-124.782,169.584,48.711,159.304
C09655=1023.011,241.132,-124.810,169.588,48.707,159.304
C09656=1023.018,241.380,-124.838,169.592,48.704,159.304
C09657=1023.023,241.628,-124.866,169.595,48.700,159.303
C09658=1023.030,241.877,-124.894,169.600,48.696,159.303
C09659=1023.036,242.125,-124.922,169.603,48.692,159.303
C09660=1023.043,242.374,-124.950,169.607,48.689,159.303
C09661=1023.049,242.622,-124.978,169.611,48.684,159.302
C09662=1023.055,242.871,-125.006,169.614,48.681,159.302
C09663=1023.061,243.119,-125.034,169.618,48.678,159.302
C09664=1023.068,243.367,-125.063,169.622,48.674,159.301
C09665=1023.074,243.615,-125.090,169.626,48.670,159.301
C09666=1023.080,243.864,-125.119,169.630,48.667,159.301
C09667=1023.087,244.113,-125.146,169.633,48.662,159.301
C09668=1023.092,244.360,-125.175,169.637,48.659,159.301
C09669=1023.098,244.609,-125.203,169.641,48.656,159.300
C09670=1023.105,244.857,-125.231,169.646,48.652,159.300
C09671=1023.111,245.105,-125.260,169.649,48.649,159.300
C09672=1023.117,245.354,-125.288,169.652,48.645,159.300
C09673=1023.124,245.602,-125.316,169.656,48.641,159.299
C09674=1023.130,245.850,-125.345,169.660,48.638,159.299
C09675=1023.136,246.099,-125.373,169.664,48.634,159.299
C09676=1023.143,246.346,-125.402,169.668,48.631,159.299
C09677=1023.149,246.595,-125.430,169.672,48.627,159.299
C09678=1023.154,246.844,-125.458,169.676,48.623,159.298
C09679=1023.162,247.138,-125.492,169.680,48.620,159.298
C09680=1023.170,247.432,-125.525,169.685,48.615,159.298
C09681=1023.177,247.726,-125.559,169.690,48.611,159.298
C09682=1023.184,248.019,-125.593,169.694,48.606,159.297
C09683=1023.195,248.434,-125.641,169.701,48.601,159.297
C09684=1023.206,248.849,-125.688,169.707,48.595,159.297
C09685=1023.216,249.265,-125.736,169.713,48.589,159.296
C09686=1023.226,249.680,-125.784,169.720,48.584,159.296
C09687=1023.233,249.928,-125.812,169.724,48.580,159.296
C09688=1023.239,250.177,-125.840,169.728,48.577,159.296
C09689=1023.245,250.425,-125.869,169.732,48.573,159.296
C09690=1023.251,250.674,-125.898,169.736,48.570,159.295
C09691=1023.258,250.922,-125.926,169.740,48.566,159.295
C09692=1023.264,251.170,-125.954,169.744,48.563,159.295
C09693=1023.270,251.418,-125.983,169.748,48.559,159.295
C09694=1023.277,251.666,-126.012,169.752,48.556,159.295
C09695=1023.283,251.915,-126.040,169.756,48.553,159.295
C09696=1023.290,252.163,-126.069,169.760,48.549,159.294
C09697=1023.296,252.411,-126.098,169.763,48.546,159.294
C09698=1023.303,252.660,-126.126,169.767,48.542,159.294
C09699=1023.309,252.908,-126.155,169.771,48.539,159.294
C09700=1023.316,253.157,-126.185,169.775,48.536,159.294
C09701=1023.322,253.405,-126.212,169.779,48.532,159.293
C09702=1023.329,253.653,-126.241,169.783,48.529,159.293
C09703=1023.335,253.901,-126.270,169.787,48.525,159.293
C09704=1023.342,254.149,-126.299,169.791,48.522,159.293
C09705=1023.348,254.398,-126.327,169.795,48.518,159.293
C09706=1023.354,254.646,-126.356,169.799,48.515,159.293
C09707=1023.360,254.894,-126.385,169.804,48.511,159.292
C09708=1023.367,255.142,-126.414,169.808,48.508,159.292
C09709=1023.373,255.391,-126.442,169.812,48.505,159.292
C09710=1023.380,255.640,-126.471,169.816,48.502,159.292
C09711=1023.387,255.887,-126.500,169.819,48.498,159.292
C09712=1023.393,256.136,-126.529,169.823,48.495,159.292
C09713=1023.400,256.384,-126.558,169.827,48.491,159.291
C09714=1023.406,256.632,-126.587,169.831,48.488,159.291
C09715=1023.413,256.880,-126.615,169.835,48.485,159.291
C09716=1023.419,257.129,-126.644,169.840,48.482,159.291
C09717=1023.426,257.377,-126.673,169.844,48.478,159.291
C09718=1023.432,257.625,-126.702,169.848,48.475,159.291
C09719=1023.439,257.873,-126.731,169.852,48.471,159.291
C09720=1023.445,258.121,-126.760,169.856,48.468,159.290
C09721=1023.452,258.370,-126.789,169.860,48.465,159.290
C09722=1023.459,258.618,-126.817,169.864,48.462,159.290
C09723=1023.465,258.866,-126.847,169.868,48.458,159.290
C09724=1023.471,259.114,-126.876,169.872,48.455,159.290
C09725=1023.478,259.363,-126.905,169.877,48.452,159.290
C09726=1023.485,259.611,-126.933,169.881,48.449,159.290
C09727=1023.492,259.859,-126.962,169.885,48.445,159.289
C09728=1023.498,260.107,-126.991,169.889,48.442,159.289
C09729=1023.505,260.355,-127.020,169.893,48.439,159.289
C09730=1023.512,260.604,-127.049,169.897,48.435,159.289
C09731=1023.518,260.852,-127.078,169.901,48.433,159.289
C09732=1023.523,261.100,-127.108,169.904,48.429,159.289
C09733=1023.530,261.348,-127.138,169.909,48.427,159.289
C09734=1023.537,261.597,-127.167,169.913,48.423,159.289
C09735=1023.543,261.845,-127.196,169.917,48.420,159.289
C09736=1023.549,262.093,-127.225,169.921,48.417,159.289
C09737=1023.556,262.341,-127.255,169.926,48.414,159.289
C09738=1023.563,262.589,-127.284,169.930,48.411,159.288
C09739=1023.573,263.003,-127.334,169.936,48.406,159.288
C09740=1023.584,263.417,-127.382,169.943,48.401,159.288
C09741=1023.595,263.831,-127.432,169.950,48.396,159.288
C09742=1023.605,264.245,-127.481,169.958,48.390,159.288
C09743=1023.612,264.493,-127.510,169.961,48.387,159.288
C09744=1023.618,264.741,-127.540,169.965,48.385,159.288
C09745=1023.624,264.990,-127.570,169.970,48.382,159.288
C09746=1023.631,265.237,-127.600,169.974,48.378,159.287
C09747=1023.637,265.485,-127.629,169.978,48.375,159.287
C09748=1023.644,265.734,-127.659,169.982,48.373,159.287
C09749=1023.651,265.982,-127.688,169.986,48.369,159.287
C09750=1023.656,266.229,-127.718,169.991,48.366,159.287
C09751=1023.663,266.478,-127.747,169.995,48.364,159.287
C09752=1023.670,266.726,-127.777,169.999,48.360,159.287
C09753=1023.676,266.975,-127.807,170.004,48.357,159.287
C09754=1023.682,267.222,-127.837,170.008,48.355,159.287
C09755=1023.689,267.471,-127.866,170.011,48.352,159.287
C09756=1023.696,267.719,-127.896,170.015,48.349,159.287
C09757=1023.702,267.967,-127.927,170.020,48.346,159.287
C09758=1023.709,268.215,-127.956,170.024,48.343,159.287
C09759=1023.715,268.463,-127.986,170.028,48.340,159.287
C09760=1023.721,268.711,-128.015,170.033,48.338,159.287
C09761=1023.728,268.960,-128.045,170.037,48.334,159.287
C09762=1023.734,269.207,-128.075,170.041,48.331,159.287
C09763=1023.741,269.456,-128.106,170.046,48.329,159.287
C09764=1023.747,269.704,-128.135,170.050,48.326,159.287
C09765=1023.754,269.952,-128.165,170.054,48.323,159.287
C09766=1023.760,270.200,-128.195,170.059,48.320,159.287
C09767=1023.767,270.447,-128.225,170.063,48.317,159.287
C09768=1023.773,270.696,-128.255,170.067,48.315,159.287
C09769=1023.779,270.944,-128.285,170.071,48.312,159.287
C09770=1023.786,271.193,-128.316,170.075,48.309,159.286
C09771=1023.792,271.440,-128.345,170.079,48.306,159.286
C09772=1023.799,271.689,-128.376,170.084,48.303,159.286
C09773=1023.805,271.936,-128.406,170.088,48.300,159.286
C09774=1023.811,272.185,-128.436,170.092,48.298,159.286
C09775=1023.818,272.433,-128.466,170.097,48.295,159.286
C09776=1023.825,272.681,-128.496,170.101,48.292,159.286
C09777=1023.831,272.929,-128.526,170.106,48.289,159.286
C09778=1023.837,273.177,-128.557,170.110,48.286,159.286
C09779=1023.844,273.425,-128.587,170.115,48.284,159.287
C09780=1023.850,273.673,-128.617,170.118,48.282,159.287
C09781=1023.857,273.922,-128.647,170.122,48.279,159.287
C09782=1023.863,274.169,-128.678,170.127,48.276,159.287
C09783=1023.870,274.418,-128.708,170.131,48.274,159.287
C09784=1023.876,274.665,-128.738,170.136,48.271,159.287
C09785=1023.883,274.914,-128.768,170.140,48.268,159.287
C09786=1023.889,275.161,-128.799,170.144,48.265,159.287
C09787=1023.896,275.409,-128.830,170.149,48.262,159.287
C09788=1023.903,275.658,-128.860,170.153,48.260,159.287
C09789=1023.909,275.905,-128.891,170.158,48.258,159.287
C09790=1023.916,276.154,-128.921,170.162,48.255,159.287
C09791=1023.922,276.401,-128.951,170.167,48.252,159.287
C09792=1023.929,276.650,-128.981,170.171,48.249,159.287
C09793=1023.935,276.898,-129.012,170.175,48.246,159.287
C09794=1023.941,277.145,-129.043,170.180,48.244,159.287
C09795=1023.953,277.564,-129.094,170.187,48.240,159.287
C09796=1023.964,277.983,-129.146,170.194,48.236,159.287
C09797=1023.974,278.401,-129.198,170.201,48.231,159.287
C09798=1023.986,278.820,-129.250,170.209,48.227,159.287
C09799=1023.992,279.067,-129.280,170.214,48.225,159.287
C09800=1023.998,279.315,-129.312,170.218,48.222,159.287
C09801=1024.005,279.564,-129.342,170.223,48.220,159.288
C09802=1024.011,279.811,-129.372,170.228,48.217,159.288
C09803=1024.018,280.059,-129.404,170.231,48.214,159.287
C09804=1024.024,280.308,-129.434,170.236,48.212,159.288
C09805=1024.030,280.555,-129.465,170.240,48.210,159.288
C09806=1024.037,280.803,-129.496,170.245,48.207,159.288
C09807=1024.044,281.051,-129.527,170.249,48.205,159.288
C09808=1024.051,281.300,-129.558,170.254,48.203,159.288
C09809=1024.057,281.547,-129.589,170.258,48.200,159.288
C09810=1024.063,281.795,-129.619,170.263,48.197,159.288
C09811=1024.070,282.043,-129.651,170.267,48.195,159.288
C09812=1024.076,282.292,-129.682,170.272,48.192,159.288
C09813=1024.083,282.539,-129.713,170.276,48.190,159.288
C09814=1024.090,282.787,-129.743,170.281,48.187,159.288
C09815=1024.096,283.035,-129.774,170.286,48.185,159.289
C09816=1024.103,283.283,-129.806,170.290,48.183,159.289
C09817=1024.110,283.532,-129.836,170.295,48.180,159.289
C09818=1024.116,283.779,-129.868,170.299,48.178,159.289
C09819=1024.122,284.027,-129.898,170.304,48.175,159.289
C09820=1024.130,284.275,-129.929,170.308,48.173,159.289
C09821=1024.136,284.523,-129.960,170.313,48.170,159.289
C09822=1024.143,284.771,-129.991,170.317,48.168,159.289
C09823=1024.149,285.019,-130.023,170.322,48.166,159.289
C09824=1024.156,285.267,-130.054,170.327,48.163,159.289
C09825=1024.162,285.514,-130.085,170.331,48.161,159.290
C09826=1024.169,285.763,-130.116,170.336,48.159,159.290
C09827=1024.175,286.011,-130.147,170.340,48.156,159.290
C09828=1024.182,286.259,-130.179,170.345,48.154,159.290
C09829=1024.189,286.506,-130.210,170.350,48.152,159.290
C09830=1024.196,286.754,-130.241,170.354,48.149,159.290
C09831=1024.202,287.002,-130.273,170.359,48.147,159.290
C09832=1024.209,287.250,-130.304,170.364,48.145,159.291
C09833=1024.216,287.498,-130.336,170.368,48.143,159.291
C09834=1024.222,287.745,-130.367,170.373,48.141,159.291
C09835=1024.228,287.994,-130.398,170.377,48.138,159.291
C09836=1024.235,288.242,-130.429,170.381,48.136,159.291
C09837=1024.242,288.490,-130.460,170.386,48.134,159.291
C09838=1024.248,288.738,-130.492,170.391,48.132,159.291
C09839=1024.255,288.985,-130.525,170.395,48.130,159.292
C09840=1024.262,289.233,-130.556,170.400,48.128,159.292
C09841=1024.268,289.481,-130.587,170.405,48.126,159.292
C09842=1024.275,289.729,-130.619,170.409,48.123,159.292
C09843=1024.282,289.977,-130.650,170.414,48.121,159.292
C09844=1024.288,290.225,-130.682,170.419,48.119,159.292
C09845=1024.294,290.473,-130.714,170.423,48.117,159.292
C09846=1024.301,290.721,-130.745,170.428,48.115,159.293
C09847=1024.308,290.969,-130.777,170.433,48.112,159.293
C09848=1024.315,291.217,-130.808,170.437,48.110,159.293
C09849=1024.322,291.464,-130.840,170.442,48.108,159.293
C09850=1024.328,291.712,-130.872,170.447,48.106,159.293
C09851=1024.334,291.927,-130.899,170.451,48.104,159.293
C09852=1024.340,292.143,-130.928,170.455,48.102,159.294
C09853=1024.345,292.358,-130.955,170.460,48.101,159.294
C09854=1024.351,292.574,-130.982,170.464,48.099,159.294
C09855=1024.357,292.788,-131.010,170.468,48.097,159.294
C09856=1024.363,293.004,-131.037,170.472,48.095,159.294
C09857=1024.368,293.219,-131.066,170.476,48.093,159.294
C09858=1024.374,293.435,-131.093,170.480,48.092,159.295
C09859=1024.381,293.682,-131.125,170.485,48.090,159.295
C09860=1024.388,293.930,-131.156,170.490,48.088,159.295
C09861=1024.394,294.178,-131.189,170.494,48.086,159.295
C09862=1024.400,294.426,-131.221,170.499,48.083,159.295
C09863=1024.407,294.673,-131.253,170.504,48.082,159.296
C09864=1024.414,294.922,-131.286,170.509,48.080,159.296
C09865=1024.421,295.169,-131.318,170.513,48.078,159.296
C09866=1024.427,295.418,-131.350,170.518,48.076,159.297
C09867=1024.433,295.665,-131.383,170.523,48.074,159.297
C09868=1024.440,295.913,-131.415,170.528,48.072,159.297
C09869=1024.446,296.161,-131.447,170.533,48.071,159.297
C09870=1024.452,296.408,-131.480,170.538,48.068,159.297
C09871=1024.459,296.656,-131.511,170.542,48.066,159.298
C09872=1024.465,296.904,-131.544,170.547,48.065,159.298
C09873=1024.473,297.152,-131.576,170.552,48.063,159.298
C09874=1024.479,297.399,-131.609,170.557,48.061,159.298
C09875=1024.485,297.648,-131.641,170.562,48.059,159.299
C09876=1024.492,297.895,-131.673,170.567,48.057,159.299
C09877=1024.499,298.143,-131.706,170.572,48.056,159.299
C09878=1024.505,298.391,-131.738,170.576,48.053,159.299
C09879=1024.512,298.639,-131.771,170.581,48.052,159.300
C09880=1024.518,298.886,-131.803,170.586,48.050,159.300
C09881=1024.525,299.134,-131.835,170.591,48.048,159.300
C09882=1024.532,299.381,-131.868,170.596,48.046,159.300
C09883=1024.539,299.629,-131.901,170.601,48.045,159.301
C09884=1024.545,299.877,-131.933,170.606,48.043,159.301
C09885=1024.552,300.125,-131.965,170.611,48.041,159.301
C09886=1024.558,300.373,-131.998,170.615,48.039,159.302
C09887=1024.566,300.621,-132.031,170.621,48.037,159.302
C09888=1024.572,300.868,-132.063,170.626,48.035,159.302
C09889=1024.578,301.116,-132.096,170.631,48.034,159.302
C09890=1024.586,301.364,-132.129,170.636,48.032,159.303
C09891=1024.592,301.611,-132.161,170.641,48.030,159.303
C09892=1024.599,301.859,-132.194,170.646,48.028,159.303
C09893=1024.606,302.107,-132.227,170.651,48.027,159.304
C09894=1024.612,302.354,-132.259,170.656,48.025,159.304
C09895=1024.619,302.602,-132.292,170.660,48.023,159.304
C09896=1024.626,302.850,-132.325,170.665,48.022,159.304
C09897=1024.633,303.098,-132.357,170.670,48.020,159.305
C09898=1024.640,303.345,-132.390,170.675,48.018,159.305
C09899=1024.646,303.593,-132.423,170.680,48.016,159.305
C09900=1024.653,303.841,-132.455,170.686,48.015,159.306
C09901=1024.660,304.089,-132.488,170.691,48.013,159.306
C09902=1024.667,304.336,-132.521,170.696,48.011,159.306
C09903=1024.674,304.585,-132.554,170.701,48.010,159.307
C09904=1024.681,304.831,-132.587,170.706,48.008,159.307
C09905=1024.687,305.079,-132.619,170.711,48.006,159.307
C09906=1024.694,305.327,-132.653,170.716,48.005,159.308
C09907=1024.701,305.575,-132.685,170.721,48.003,159.308
C09908=1024.708,305.823,-132.718,170.727,48.001,159.308
C09909=1024.715,306.069,-132.751,170.732,47.999,159.308
C09910=1024.722,306.318,-132.784,170.737,47.998,159.309
C09911=1024.728,306.542,-132.814,170.741,47.997,159.309
C09912=1024.734,306.766,-132.843,170.746,47.995,159.309
C09913=1024.740,306.990,-132.873,170.751,47.994,159.310
C09914=1024.747,307.213,-132.903,170.754,47.992,159.310
C09915=1024.753,307.438,-132.932,170.759,47.990,159.310
C09916=1024.760,307.662,-132.963,170.765,47.989,159.311
C09917=1024.766,307.886,-132.993,170.769,47.988,159.311
C09918=1024.772,308.110,-133.023,170.774,47.986,159.311
C09919=1024.780,308.358,-133.055,170.779,47.985,159.312
C09920=1024.786,308.605,-133.088,170.784,47.983,159.312
C09921=1024.793,308.853,-133.122,170.790,47.982,159.312
C09922=1024.800,309.100,-133.154,170.795,47.980,159.313
C09923=1024.808,309.348,-133.188,170.800,47.979,159.313
C09924=1024.815,309.596,-133.221,170.804,47.976,159.313
C09925=1024.822,309.843,-133.254,170.810,47.975,159.314
C09926=1024.829,310.091,-133.287,170.816,47.973,159.314
C09927=1024.836,310.339,-133.321,170.821,47.972,159.314
C09928=1024.843,310.586,-133.353,170.826,47.970,159.315
C09929=1024.849,310.834,-133.387,170.831,47.969,159.315
C09930=1024.856,311.081,-133.421,170.836,47.968,159.316
C09931=1024.863,311.329,-133.455,170.841,47.967,159.316
C09932=1024.870,311.577,-133.488,170.846,47.965,159.316
C09933=1024.876,311.824,-133.522,170.851,47.964,159.317
C09934=1024.883,312.072,-133.556,170.858,47.962,159.317
C09935=1024.890,312.319,-133.589,170.863,47.961,159.318
C09936=1024.896,312.567,-133.623,170.868,47.960,159.318
C09937=1024.903,312.815,-133.657,170.873,47.959,159.319
C09938=1024.910,313.062,-133.691,170.878,47.957,159.319
C09939=1024.917,313.310,-133.725,170.883,47.956,159.320
C09940=1024.924,313.557,-133.759,170.888,47.955,159.320
C09941=1024.930,313.804,-133.792,170.894,47.953,159.320
C09942=1024.938,314.052,-133.826,170.900,47.952,159.321
C09943=1024.944,314.300,-133.861,170.905,47.951,159.321
C09944=1024.951,314.548,-133.895,170.910,47.950,159.322
C09945=1024.958,314.794,-133.928,170.915,47.948,159.322
C09946=1024.964,315.042,-133.962,170.920,47.947,159.322
C09947=1024.971,315.290,-133.996,170.927,47.946,159.323
C09948=1024.979,315.538,-134.030,170.932,47.944,159.323
C09949=1024.985,315.785,-134.064,170.937,47.944,159.324
C09950=1024.992,316.033,-134.098,170.942,47.942,159.324
C09951=1024.999,316.280,-134.132,170.947,47.941,159.325
C09952=1025.006,316.528,-134.166,170.954,47.939,159.325
C09953=1025.013,316.775,-134.201,170.959,47.939,159.326
C09954=1025.020,317.023,-134.235,170.964,47.937,159.326
C09955=1025.027,317.270,-134.268,170.969,47.936,159.327
C09956=1025.033,317.518,-134.302,170.975,47.936,159.327
C09957=1025.040,317.766,-134.336,170.981,47.934,159.328
C09958=1025.048,318.013,-134.371,170.986,47.933,159.328
C09959=1025.054,318.261,-134.405,170.991,47.931,159.329
C09960=1025.062,318.509,-134.439,170.996,47.931,159.329
C09961=1025.069,318.756,-134.474,171.002,47.930,159.330
C09962=1025.075,319.004,-134.508,171.008,47.928,159.330
C09963=1025.083,319.251,-134.542,171.013,47.927,159.331
C09964=1025.090,319.498,-134.576,171.019,47.926,159.331
C09965=1025.097,319.746,-134.611,171.024,47.925,159.332
C09966=1025.104,319.994,-134.645,171.030,47.924,159.332
C09967=1025.111,320.241,-134.679,171.035,47.923,159.333
C09968=1025.118,320.489,-134.714,171.040,47.921,159.333
C09969=1025.125,320.736,-134.748,171.047,47.920,159.334
C09970=1025.133,320.984,-134.782,171.052,47.919,159.334
C09971=1025.138,321.210,-134.813,171.057,47.918,159.335
C09972=1025.145,321.436,-134.845,171.062,47.917,159.335
C09973=1025.151,321.664,-134.877,171.067,47.917,159.336
C09974=1025.158,321.889,-134.908,171.072,47.916,159.336
C09975=1025.165,322.116,-134.939,171.077,47.914,159.336
C09976=1025.171,322.343,-134.971,171.083,47.913,159.337
C09977=1025.178,322.569,-135.003,171.088,47.913,159.338
C09978=1025.184,322.796,-135.034,171.093,47.912,159.338
C09979=1025.192,323.044,-135.069,171.099,47.911,159.339
C09980=1025.200,323.291,-135.103,171.104,47.909,159.339
C09981=1025.206,323.539,-135.138,171.110,47.908,159.340
C09982=1025.214,323.786,-135.172,171.115,47.907,159.340
C09983=1025.220,324.034,-135.207,171.121,47.907,159.341
C09984=1025.228,324.281,-135.241,171.127,47.905,159.341
C09985=1025.236,324.528,-135.276,171.133,47.905,159.342
C09986=1025.242,324.776,-135.311,171.138,47.904,159.342
C09987=1025.250,325.024,-135.345,171.144,47.903,159.343
C09988=1025.257,325.271,-135.380,171.150,47.902,159.343
C09989=1025.264,325.519,-135.415,171.155,47.901,159.344
C09990=1025.272,325.766,-135.450,171.161,47.900,159.345
C09991=1025.279,326.013,-135.483,171.167,47.899,159.345
C09992=1025.286,326.261,-135.519,171.173,47.898,159.346
C09993=1025.294,326.508,-135.554,171.178,47.897,159.346
C09994=1025.301,326.756,-135.589,171.184,47.896,159.347
C09995=1025.308,327.003,-135.623,171.190,47.895,159.347
C09996=1025.316,327.250,-135.658,171.195,47.894,159.348
//INST
///DATE 2021/06/17 10:59
///ATTR SC,RW,RJ
////FRAME ROBOT
///GROUP1 RB1
NOP
MOVL C00000 V=800.0 PL=0
MOVL C00001 V=800.0 PL=0
MOVL C00002 V=800.0 PL=0
MOVL C00003 V=800.0 PL=0
MOVL C00004 V=800.0 PL=0
MOVL C00005 V=800.0 PL=0
MOVL C00006 V=800.0 PL=0
MOVL C00007 V=800.0 PL=0
MOVL C00008 V=800.0 PL=0
MOVL C00009 V=800.0 PL=0
MOVL C00010 V=800.0 PL=0
MOVL C00011 V=800.0 PL=0
MOVL C00012 V=800.0 PL=0
MOVL C00013 V=800.0 PL=0
MOVL C00014 V=800.0 PL=0
MOVL C00015 V=800.0 PL=0
MOVL C00016 V=800.0 PL=0
MOVL C00017 V=800.0 PL=0
MOVL C00018 V=800.0 PL=0
MOVL C00019 V=800.0 PL=0
MOVL C00020 V=800.0 PL=0
MOVL C00021 V=800.0 PL=0
MOVL C00022 V=800.0 PL=0
MOVL C00023 V=800.0 PL=0
MOVL C00024 V=800.0 PL=0
MOVL C00025 V=800.0 PL=0
MOVL C00026 V=800.0 PL=0
MOVL C00027 V=800.0 PL=0
MOVL C00028 V=800.0 PL=0
MOVL C00029 V=800.0 PL=0
MOVL C00030 V=800.0 PL=0
MOVL C00031 V=800.0 PL=0
MOVL C00032 V=800.0 PL=0
MOVL C00033 V=800.0 PL=0
MOVL C00034 V=800.0 PL=0
MOVL C00035 V=800.0 PL=0
MOVL C00036 V=800.0 PL=0
MOVL C00037 V=800.0 PL=0
MOVL C00038 V=800.0 PL=0
MOVL C00039 V=800.0 PL=0
MOVL C00040 V=800.0 PL=0
MOVL C00041 V=800.0 PL=0
MOVL C00042 V=800.0 PL=0
MOVL C00043 V=800.0 PL=0
MOVL C00044 V=800.0 PL=0
MOVL C00045 V=800.0 PL=0
MOVL C00046 V=800.0 PL=0
MOVL C00047 V=800.0 PL=0
MOVL C00048 V=800.0 PL=0
MOVL C00049 V=800.0 PL=0
MOVL C00050 V=800.0 PL=0
MOVL C00051 V=800.0 PL=0
MOVL C00052 V=800.0 PL=0
MOVL C00053 V=800.0 PL=0
MOVL C00054 V=800.0 PL=0
MOVL C00055 V=800.0 PL=0
MOVL C00056 V=800.0 PL=0
MOVL C00057 V=800.0 PL=0
MOVL C00058 V=800.0 PL=0
MOVL C00059 V=800.0 PL=0
MOVL C00060 V=800.0 PL=0
MOVL C00061 V=800.0 PL=0
MOVL C00062 V=800.0 PL=0
MOVL C00063 V=800.0 PL=0
MOVL C00064 V=800.0 PL=0
MOVL C00065 V=800.0 PL=0
MOVL C00066 V=800.0 PL=0
MOVL C00067 V=800.0 PL=0
MOVL C00068 V=800.0 PL=0
MOVL C00069 V=800.0 PL=0
MOVL C00070 V=800.0 PL=0
MOVL C00071 V=800.0 PL=0
MOVL C00072 V=800.0 PL=0
MOVL C00073 V=800.0 PL=0
MOVL C00074 V=800.0 PL=0
MOVL C00075 V=800.0 PL=0
MOVL C00076 V=800.0 PL=0
MOVL C00077 V=800.0 PL=0
MOVL C00078 V=800.0 PL=0
MOVL C00079 V=800.0 PL=0
MOVL C00080 V=800.0 PL=0
MOVL C00081 V=800.0 PL=0
MOVL C00082 V=800.0 PL=0
MOVL C00083 V=800.0 PL=0
MOVL C00084 V=800.0 PL=0
MOVL C00085 V=800.0 PL=0
MOVL C00086 V=800.0 PL=0
MOVL C00087 V=800.0 PL=0
MOVL C00088 V=800.0 PL=0
MOVL C00089 V=800.0 PL=0
MOVL C00090 V=800.0 PL=0
MOVL C00091 V=800.0 PL=0
MOVL C00092 V=800.0 PL=0
MOVL C00093 V=800.0 PL=0
MOVL C00094 V=800.0 PL=0
MOVL C00095 V=800.0 PL=0
MOVL C00096 V=800.0 PL=0
MOVL C00097 V=800.0 PL=0
MOVL C00098 V=800.0 PL=0
MOVL C00099 V=800.0 PL=0
MOVL C00100 V=800.0 PL=0
MOVL C00101 V=800.0 PL=0
MOVL C00102 V=800.0 PL=0
MOVL C00103 V=800.0 PL=0
MOVL C00104 V=800.0 PL=0
MOVL C00105 V=800.0 PL=0
MOVL C00106 V=800.0 PL=0
MOVL C00107 V=800.0 PL=0
MOVL C00108 V=800.0 PL=0
MOVL C00109 V=800.0 PL=0
MOVL C00110 V=800.0 PL=0
MOVL C00111 V=800.0 PL=0
MOVL C00112 V=800.0 PL=0
MOVL C00113 V=800.0 PL=0
MOVL C00114 V=800.0 PL=0
MOVL C00115 V=800.0 PL=0
MOVL C00116 V=800.0 PL=0
MOVL C00117 V=800.0 PL=0
MOVL C00118 V=800.0 PL=0
MOVL C00119 V=800.0 PL=0
MOVL C00120 V=800.0 PL=0
MOVL C00121 V=800.0 PL=0
MOVL C00122 V=800.0 PL=0
MOVL C00123 V=800.0 PL=0
MOVL C00124 V=800.0 PL=0
MOVL C00125 V=800.0 PL=0
MOVL C00126 V=800.0 PL=0
MOVL C00127 V=800.0 PL=0
MOVL C00128 V=800.0 PL=0
MOVL C00129 V=800.0 PL=0
MOVL C00130 V=800.0 PL=0
MOVL C00131 V=800.0 PL=0
MOVL C00132 V=800.0 PL=0
MOVL C00133 V=800.0 PL=0
MOVL C00134 V=800.0 PL=0
MOVL C00135 V=800.0 PL=0
MOVL C00136 V=800.0 PL=0
MOVL C00137 V=800.0 PL=0
MOVL C00138 V=800.0 PL=0
MOVL C00139 V=800.0 PL=0
MOVL C00140 V=800.0 PL=0
MOVL C00141 V=800.0 PL=0
MOVL C00142 V=800.0 PL=0
MOVL C00143 V=800.0 PL=0
MOVL C00144 V=800.0 PL=0
MOVL C00145 V=800.0 PL=0
MOVL C00146 V=800.0 PL=0
MOVL C00147 V=800.0 PL=0
MOVL C00148 V=800.0 PL=0
MOVL C00149 V=800.0 PL=0
MOVL C00150 V=800.0 PL=0
MOVL C00151 V=800.0 PL=0
MOVL C00152 V=800.0 PL=0
MOVL C00153 V=800.0 PL=0
MOVL C00154 V=800.0 PL=0
MOVL C00155 V=800.0 PL=0
MOVL C00156 V=800.0 PL=0
MOVL C00157 V=800.0 PL=0
MOVL C00158 V=800.0 PL=0
MOVL C00159 V=800.0 PL=0
MOVL C00160 V=800.0 PL=0
MOVL C00161 V=800.0 PL=0
MOVL C00162 V=800.0 PL=0
MOVL C00163 V=800.0 PL=0
MOVL C00164 V=800.0 PL=0
MOVL C00165 V=800.0 PL=0
MOVL C00166 V=800.0 PL=0
MOVL C00167 V=800.0 PL=0
MOVL C00168 V=800.0 PL=0
MOVL C00169 V=800.0 PL=0
MOVL C00170 V=800.0 PL=0
MOVL C00171 V=800.0 PL=0
MOVL C00172 V=800.0 PL=0
MOVL C00173 V=800.0 PL=0
MOVL C00174 V=800.0 PL=0
MOVL C00175 V=800.0 PL=0
MOVL C00176 V=800.0 PL=0
MOVL C00177 V=800.0 PL=0
MOVL C00178 V=800.0 PL=0
MOVL C00179 V=800.0 PL=0
MOVL C00180 V=800.0 PL=0
MOVL C00181 V=800.0 PL=0
MOVL C00182 V=800.0 PL=0
MOVL C00183 V=800.0 PL=0
MOVL C00184 V=800.0 PL=0
MOVL C00185 V=800.0 PL=0
MOVL C00186 V=800.0 PL=0
MOVL C00187 V=800.0 PL=0
MOVL C00188 V=800.0 PL=0
MOVL C00189 V=800.0 PL=0
MOVL C00190 V=800.0 PL=0
MOVL C00191 V=800.0 PL=0
MOVL C00192 V=800.0 PL=0
MOVL C00193 V=800.0 PL=0
MOVL C00194 V=800.0 PL=0
MOVL C00195 V=800.0 PL=0
MOVL C00196 V=800.0 PL=0
MOVL C00197 V=800.0 PL=0
MOVL C00198 V=800.0 PL=0
MOVL C00199 V=800.0 PL=0
MOVL C00200 V=800.0 PL=0
MOVL C00201 V=800.0 PL=0
MOVL C00202 V=800.0 PL=0
MOVL C00203 V=800.0 PL=0
MOVL C00204 V=800.0 PL=0
MOVL C00205 V=800.0 PL=0
MOVL C00206 V=800.0 PL=0
MOVL C00207 V=800.0 PL=0
MOVL C00208 V=800.0 PL=0
MOVL C00209 V=800.0 PL=0
MOVL C00210 V=800.0 PL=0
MOVL C00211 V=800.0 PL=0
MOVL C00212 V=800.0 PL=0
MOVL C00213 V=800.0 PL=0
MOVL C00214 V=800.0 PL=0
MOVL C00215 V=800.0 PL=0
MOVL C00216 V=800.0 PL=0
MOVL C00217 V=800.0 PL=0
MOVL C00218 V=800.0 PL=0
MOVL C00219 V=800.0 PL=0
MOVL C00220 V=800.0 PL=0
MOVL C00221 V=800.0 PL=0
MOVL C00222 V=800.0 PL=0
MOVL C00223 V=800.0 PL=0
MOVL C00224 V=800.0 PL=0
MOVL C00225 V=800.0 PL=0
MOVL C00226 V=800.0 PL=0
MOVL C00227 V=800.0 PL=0
MOVL C00228 V=800.0 PL=0
MOVL C00229 V=800.0 PL=0
MOVL C00230 V=800.0 PL=0
MOVL C00231 V=800.0 PL=0
MOVL C00232 V=800.0 PL=0
MOVL C00233 V=800.0 PL=0
MOVL C00234 V=800.0 PL=0
MOVL C00235 V=800.0 PL=0
MOVL C00236 V=800.0 PL=0
MOVL C00237 V=800.0 PL=0
MOVL C00238 V=800.0 PL=0
MOVL C00239 V=800.0 PL=0
MOVL C00240 V=800.0 PL=0
MOVL C00241 V=800.0 PL=0
MOVL C00242 V=800.0 PL=0
MOVL C00243 V=800.0 PL=0
MOVL C00244 V=800.0 PL=0
MOVL C00245 V=800.0 PL=0
MOVL C00246 V=800.0 PL=0
MOVL C00247 V=800.0 PL=0
MOVL C00248 V=800.0 PL=0
MOVL C00249 V=800.0 PL=0
MOVL C00250 V=800.0 PL=0
MOVL C00251 V=800.0 PL=0
MOVL C00252 V=800.0 PL=0
MOVL C00253 V=800.0 PL=0
MOVL C00254 V=800.0 PL=0
MOVL C00255 V=800.0 PL=0
MOVL C00256 V=800.0 PL=0
MOVL C00257 V=800.0 PL=0
MOVL C00258 V=800.0 PL=0
MOVL C00259 V=800.0 PL=0
MOVL C00260 V=800.0 PL=0
MOVL C00261 V=800.0 PL=0
MOVL C00262 V=800.0 PL=0
MOVL C00263 V=800.0 PL=0
MOVL C00264 V=800.0 PL=0
MOVL C00265 V=800.0 PL=0
MOVL C00266 V=800.0 PL=0
MOVL C00267 V=800.0 PL=0
MOVL C00268 V=800.0 PL=0
MOVL C00269 V=800.0 PL=0
MOVL C00270 V=800.0 PL=0
MOVL C00271 V=800.0 PL=0
MOVL C00272 V=800.0 PL=0
MOVL C00273 V=800.0 PL=0
MOVL C00274 V=800.0 PL=0
MOVL C00275 V=800.0 PL=0
MOVL C00276 V=800.0 PL=0
MOVL C00277 V=800.0 PL=0
MOVL C00278 V=800.0 PL=0
MOVL C00279 V=800.0 PL=0
MOVL C00280 V=800.0 PL=0
MOVL C00281 V=800.0 PL=0
MOVL C00282 V=800.0 PL=0
MOVL C00283 V=800.0 PL=0
MOVL C00284 V=800.0 PL=0
MOVL C00285 V=800.0 PL=0
MOVL C00286 V=800.0 PL=0
MOVL C00287 V=800.0 PL=0
MOVL C00288 V=800.0 PL=0
MOVL C00289 V=800.0 PL=0
MOVL C00290 V=800.0 PL=0
MOVL C00291 V=800.0 PL=0
MOVL C00292 V=800.0 PL=0
MOVL C00293 V=800.0 PL=0
MOVL C00294 V=800.0 PL=0
MOVL C00295 V=800.0 PL=0
MOVL C00296 V=800.0 PL=0
MOVL C00297 V=800.0 PL=0
MOVL C00298 V=800.0 PL=0
MOVL C00299 V=800.0 PL=0
MOVL C00300 V=800.0 PL=0
MOVL C00301 V=800.0 PL=0
MOVL C00302 V=800.0 PL=0
MOVL C00303 V=800.0 PL=0
MOVL C00304 V=800.0 PL=0
MOVL C00305 V=800.0 PL=0
MOVL C00306 V=800.0 PL=0
MOVL C00307 V=800.0 PL=0
MOVL C00308 V=800.0 PL=0
MOVL C00309 V=800.0 PL=0
MOVL C00310 V=800.0 PL=0
MOVL C00311 V=800.0 PL=0
MOVL C00312 V=800.0 PL=0
MOVL C00313 V=800.0 PL=0
MOVL C00314 V=800.0 PL=0
MOVL C00315 V=800.0 PL=0
MOVL C00316 V=800.0 PL=0
MOVL C00317 V=800.0 PL=0
MOVL C00318 V=800.0 PL=0
MOVL C00319 V=800.0 PL=0
MOVL C00320 V=800.0 PL=0
MOVL C00321 V=800.0 PL=0
MOVL C00322 V=800.0 PL=0
MOVL C00323 V=800.0 PL=0
MOVL C00324 V=800.0 PL=0
MOVL C00325 V=800.0 PL=0
MOVL C00326 V=800.0 PL=0
MOVL C00327 V=800.0 PL=0
MOVL C00328 V=800.0 PL=0
MOVL C00329 V=800.0 PL=0
MOVL C00330 V=800.0 PL=0
MOVL C00331 V=800.0 PL=0
MOVL C00332 V=800.0 PL=0
MOVL C00333 V=800.0 PL=0
MOVL C00334 V=800.0 PL=0
MOVL C00335 V=800.0 PL=0
MOVL C00336 V=800.0 PL=0
MOVL C00337 V=800.0 PL=0
MOVL C00338 V=800.0 PL=0
MOVL C00339 V=800.0 PL=0
MOVL C00340 V=800.0 PL=0
MOVL C00341 V=800.0 PL=0
MOVL C00342 V=800.0 PL=0
MOVL C00343 V=800.0 PL=0
MOVL C00344 V=800.0 PL=0
MOVL C00345 V=800.0 PL=0
MOVL C00346 V=800.0 PL=0
MOVL C00347 V=800.0 PL=0
MOVL C00348 V=800.0 PL=0
MOVL C00349 V=800.0 PL=0
MOVL C00350 V=800.0 PL=0
MOVL C00351 V=800.0 PL=0
MOVL C00352 V=800.0 PL=0
MOVL C00353 V=800.0 PL=0
MOVL C00354 V=800.0 PL=0
MOVL C00355 V=800.0 PL=0
MOVL C00356 V=800.0 PL=0
MOVL C00357 V=800.0 PL=0
MOVL C00358 V=800.0 PL=0
MOVL C00359 V=800.0 PL=0
MOVL C00360 V=800.0 PL=0
MOVL C00361 V=800.0 PL=0
MOVL C00362 V=800.0 PL=0
MOVL C00363 V=800.0 PL=0
MOVL C00364 V=800.0 PL=0
MOVL C00365 V=800.0 PL=0
MOVL C00366 V=800.0 PL=0
MOVL C00367 V=800.0 PL=0
MOVL C00368 V=800.0 PL=0
MOVL C00369 V=800.0 PL=0
MOVL C00370 V=800.0 PL=0
MOVL C00371 V=800.0 PL=0
MOVL C00372 V=800.0 PL=0
MOVL C00373 V=800.0 PL=0
MOVL C00374 V=800.0 PL=0
MOVL C00375 V=800.0 PL=0
MOVL C00376 V=800.0 PL=0
MOVL C00377 V=800.0 PL=0
MOVL C00378 V=800.0 PL=0
MOVL C00379 V=800.0 PL=0
MOVL C00380 V=800.0 PL=0
MOVL C00381 V=800.0 PL=0
MOVL C00382 V=800.0 PL=0
MOVL C00383 V=800.0 PL=0
MOVL C00384 V=800.0 PL=0
MOVL C00385 V=800.0 PL=0
MOVL C00386 V=800.0 PL=0
MOVL C00387 V=800.0 PL=0
MOVL C00388 V=800.0 PL=0
MOVL C00389 V=800.0 PL=0
MOVL C00390 V=800.0 PL=0
MOVL C00391 V=800.0 PL=0
MOVL C00392 V=800.0 PL=0
MOVL C00393 V=800.0 PL=0
MOVL C00394 V=800.0 PL=0
MOVL C00395 V=800.0 PL=0
MOVL C00396 V=800.0 PL=0
MOVL C00397 V=800.0 PL=0
MOVL C00398 V=800.0 PL=0
MOVL C00399 V=800.0 PL=0
MOVL C00400 V=800.0 PL=0
MOVL C00401 V=800.0 PL=0
MOVL C00402 V=800.0 PL=0
MOVL C00403 V=800.0 PL=0
MOVL C00404 V=800.0 PL=0
MOVL C00405 V=800.0 PL=0
MOVL C00406 V=800.0 PL=0
MOVL C00407 V=800.0 PL=0
MOVL C00408 V=800.0 PL=0
MOVL C00409 V=800.0 PL=0
MOVL C00410 V=800.0 PL=0
MOVL C00411 V=800.0 PL=0
MOVL C00412 V=800.0 PL=0
MOVL C00413 V=800.0 PL=0
MOVL C00414 V=800.0 PL=0
MOVL C00415 V=800.0 PL=0
MOVL C00416 V=800.0 PL=0
MOVL C00417 V=800.0 PL=0
MOVL C00418 V=800.0 PL=0
MOVL C00419 V=800.0 PL=0
MOVL C00420 V=800.0 PL=0
MOVL C00421 V=800.0 PL=0
MOVL C00422 V=800.0 PL=0
MOVL C00423 V=800.0 PL=0
MOVL C00424 V=800.0 PL=0
MOVL C00425 V=800.0 PL=0
MOVL C00426 V=800.0 PL=0
MOVL C00427 V=800.0 PL=0
MOVL C00428 V=800.0 PL=0
MOVL C00429 V=800.0 PL=0
MOVL C00430 V=800.0 PL=0
MOVL C00431 V=800.0 PL=0
MOVL C00432 V=800.0 PL=0
MOVL C00433 V=800.0 PL=0
MOVL C00434 V=800.0 PL=0
MOVL C00435 V=800.0 PL=0
MOVL C00436 V=800.0 PL=0
MOVL C00437 V=800.0 PL=0
MOVL C00438 V=800.0 PL=0
MOVL C00439 V=800.0 PL=0
MOVL C00440 V=800.0 PL=0
MOVL C00441 V=800.0 PL=0
MOVL C00442 V=800.0 PL=0
MOVL C00443 V=800.0 PL=0
MOVL C00444 V=800.0 PL=0
MOVL C00445 V=800.0 PL=0
MOVL C00446 V=800.0 PL=0
MOVL C00447 V=800.0 PL=0
MOVL C00448 V=800.0 PL=0
MOVL C00449 V=800.0 PL=0
MOVL C00450 V=800.0 PL=0
MOVL C00451 V=800.0 PL=0
MOVL C00452 V=800.0 PL=0
MOVL C00453 V=800.0 PL=0
MOVL C00454 V=800.0 PL=0
MOVL C00455 V=800.0 PL=0
MOVL C00456 V=800.0 PL=0
MOVL C00457 V=800.0 PL=0
MOVL C00458 V=800.0 PL=0
MOVL C00459 V=800.0 PL=0
MOVL C00460 V=800.0 PL=0
MOVL C00461 V=800.0 PL=0
MOVL C00462 V=800.0 PL=0
MOVL C00463 V=800.0 PL=0
MOVL C00464 V=800.0 PL=0
MOVL C00465 V=800.0 PL=0
MOVL C00466 V=800.0 PL=0
MOVL C00467 V=800.0 PL=0
MOVL C00468 V=800.0 PL=0
MOVL C00469 V=800.0 PL=0
MOVL C00470 V=800.0 PL=0
MOVL C00471 V=800.0 PL=0
MOVL C00472 V=800.0 PL=0
MOVL C00473 V=800.0 PL=0
MOVL C00474 V=800.0 PL=0
MOVL C00475 V=800.0 PL=0
MOVL C00476 V=800.0 PL=0
MOVL C00477 V=800.0 PL=0
MOVL C00478 V=800.0 PL=0
MOVL C00479 V=800.0 PL=0
MOVL C00480 V=800.0 PL=0
MOVL C00481 V=800.0 PL=0
MOVL C00482 V=800.0 PL=0
MOVL C00483 V=800.0 PL=0
MOVL C00484 V=800.0 PL=0
MOVL C00485 V=800.0 PL=0
MOVL C00486 V=800.0 PL=0
MOVL C00487 V=800.0 PL=0
MOVL C00488 V=800.0 PL=0
MOVL C00489 V=800.0 PL=0
MOVL C00490 V=800.0 PL=0
MOVL C00491 V=800.0 PL=0
MOVL C00492 V=800.0 PL=0
MOVL C00493 V=800.0 PL=0
MOVL C00494 V=800.0 PL=0
MOVL C00495 V=800.0 PL=0
MOVL C00496 V=800.0 PL=0
MOVL C00497 V=800.0 PL=0
MOVL C00498 V=800.0 PL=0
MOVL C00499 V=800.0 PL=0
MOVL C00500 V=800.0 PL=0
MOVL C00501 V=800.0 PL=0
MOVL C00502 V=800.0 PL=0
MOVL C00503 V=800.0 PL=0
MOVL C00504 V=800.0 PL=0
MOVL C00505 V=800.0 PL=0
MOVL C00506 V=800.0 PL=0
MOVL C00507 V=800.0 PL=0
MOVL C00508 V=800.0 PL=0
MOVL C00509 V=800.0 PL=0
MOVL C00510 V=800.0 PL=0
MOVL C00511 V=800.0 PL=0
MOVL C00512 V=800.0 PL=0
MOVL C00513 V=800.0 PL=0
MOVL C00514 V=800.0 PL=0
MOVL C00515 V=800.0 PL=0
MOVL C00516 V=800.0 PL=0
MOVL C00517 V=800.0 PL=0
MOVL C00518 V=800.0 PL=0
MOVL C00519 V=800.0 PL=0
MOVL C00520 V=800.0 PL=0
MOVL C00521 V=800.0 PL=0
MOVL C00522 V=800.0 PL=0
MOVL C00523 V=800.0 PL=0
MOVL C00524 V=800.0 PL=0
MOVL C00525 V=800.0 PL=0
MOVL C00526 V=800.0 PL=0
MOVL C00527 V=800.0 PL=0
MOVL C00528 V=800.0 PL=0
MOVL C00529 V=800.0 PL=0
MOVL C00530 V=800.0 PL=0
MOVL C00531 V=800.0 PL=0
MOVL C00532 V=800.0 PL=0
MOVL C00533 V=800.0 PL=0
MOVL C00534 V=800.0 PL=0
MOVL C00535 V=800.0 PL=0
MOVL C00536 V=800.0 PL=0
MOVL C00537 V=800.0 PL=0
MOVL C00538 V=800.0 PL=0
MOVL C00539 V=800.0 PL=0
MOVL C00540 V=800.0 PL=0
MOVL C00541 V=800.0 PL=0
MOVL C00542 V=800.0 PL=0
MOVL C00543 V=800.0 PL=0
MOVL C00544 V=800.0 PL=0
MOVL C00545 V=800.0 PL=0
MOVL C00546 V=800.0 PL=0
MOVL C00547 V=800.0 PL=0
MOVL C00548 V=800.0 PL=0
MOVL C00549 V=800.0 PL=0
MOVL C00550 V=800.0 PL=0
MOVL C00551 V=800.0 PL=0
MOVL C00552 V=800.0 PL=0
MOVL C00553 V=800.0 PL=0
MOVL C00554 V=800.0 PL=0
MOVL C00555 V=800.0 PL=0
MOVL C00556 V=800.0 PL=0
MOVL C00557 V=800.0 PL=0
MOVL C00558 V=800.0 PL=0
MOVL C00559 V=800.0 PL=0
MOVL C00560 V=800.0 PL=0
MOVL C00561 V=800.0 PL=0
MOVL C00562 V=800.0 PL=0
MOVL C00563 V=800.0 PL=0
MOVL C00564 V=800.0 PL=0
MOVL C00565 V=800.0 PL=0
MOVL C00566 V=800.0 PL=0
MOVL C00567 V=800.0 PL=0
MOVL C00568 V=800.0 PL=0
MOVL C00569 V=800.0 PL=0
MOVL C00570 V=800.0 PL=0
MOVL C00571 V=800.0 PL=0
MOVL C00572 V=800.0 PL=0
MOVL C00573 V=800.0 PL=0
MOVL C00574 V=800.0 PL=0
MOVL C00575 V=800.0 PL=0
MOVL C00576 V=800.0 PL=0
MOVL C00577 V=800.0 PL=0
MOVL C00578 V=800.0 PL=0
MOVL C00579 V=800.0 PL=0
MOVL C00580 V=800.0 PL=0
MOVL C00581 V=800.0 PL=0
MOVL C00582 V=800.0 PL=0
MOVL C00583 V=800.0 PL=0
MOVL C00584 V=800.0 PL=0
MOVL C00585 V=800.0 PL=0
MOVL C00586 V=800.0 PL=0
MOVL C00587 V=800.0 PL=0
MOVL C00588 V=800.0 PL=0
MOVL C00589 V=800.0 PL=0
MOVL C00590 V=800.0 PL=0
MOVL C00591 V=800.0 PL=0
MOVL C00592 V=800.0 PL=0
MOVL C00593 V=800.0 PL=0
MOVL C00594 V=800.0 PL=0
MOVL C00595 V=800.0 PL=0
MOVL C00596 V=800.0 PL=0
MOVL C00597 V=800.0 PL=0
MOVL C00598 V=800.0 PL=0
MOVL C00599 V=800.0 PL=0
MOVL C00600 V=800.0 PL=0
MOVL C00601 V=800.0 PL=0
MOVL C00602 V=800.0 PL=0
MOVL C00603 V=800.0 PL=0
MOVL C00604 V=800.0 PL=0
MOVL C00605 V=800.0 PL=0
MOVL C00606 V=800.0 PL=0
MOVL C00607 V=800.0 PL=0
MOVL C00608 V=800.0 PL=0
MOVL C00609 V=800.0 PL=0
MOVL C00610 V=800.0 PL=0
MOVL C00611 V=800.0 PL=0
MOVL C00612 V=800.0 PL=0
MOVL C00613 V=800.0 PL=0
MOVL C00614 V=800.0 PL=0
MOVL C00615 V=800.0 PL=0
MOVL C00616 V=800.0 PL=0
MOVL C00617 V=800.0 PL=0
MOVL C00618 V=800.0 PL=0
MOVL C00619 V=800.0 PL=0
MOVL C00620 V=800.0 PL=0
MOVL C00621 V=800.0 PL=0
MOVL C00622 V=800.0 PL=0
MOVL C00623 V=800.0 PL=0
MOVL C00624 V=800.0 PL=0
MOVL C00625 V=800.0 PL=0
MOVL C00626 V=800.0 PL=0
MOVL C00627 V=800.0 PL=0
MOVL C00628 V=800.0 PL=0
MOVL C00629 V=800.0 PL=0
MOVL C00630 V=800.0 PL=0
MOVL C00631 V=800.0 PL=0
MOVL C00632 V=800.0 PL=0
MOVL C00633 V=800.0 PL=0
MOVL C00634 V=800.0 PL=0
MOVL C00635 V=800.0 PL=0
MOVL C00636 V=800.0 PL=0
MOVL C00637 V=800.0 PL=0
MOVL C00638 V=800.0 PL=0
MOVL C00639 V=800.0 PL=0
MOVL C00640 V=800.0 PL=0
MOVL C00641 V=800.0 PL=0
MOVL C00642 V=800.0 PL=0
MOVL C00643 V=800.0 PL=0
MOVL C00644 V=800.0 PL=0
MOVL C00645 V=800.0 PL=0
MOVL C00646 V=800.0 PL=0
MOVL C00647 V=800.0 PL=0
MOVL C00648 V=800.0 PL=0
MOVL C00649 V=800.0 PL=0
MOVL C00650 V=800.0 PL=0
MOVL C00651 V=800.0 PL=0
MOVL C00652 V=800.0 PL=0
MOVL C00653 V=800.0 PL=0
MOVL C00654 V=800.0 PL=0
MOVL C00655 V=800.0 PL=0
MOVL C00656 V=800.0 PL=0
MOVL C00657 V=800.0 PL=0
MOVL C00658 V=800.0 PL=0
MOVL C00659 V=800.0 PL=0
MOVL C00660 V=800.0 PL=0
MOVL C00661 V=800.0 PL=0
MOVL C00662 V=800.0 PL=0
MOVL C00663 V=800.0 PL=0
MOVL C00664 V=800.0 PL=0
MOVL C00665 V=800.0 PL=0
MOVL C00666 V=800.0 PL=0
MOVL C00667 V=800.0 PL=0
MOVL C00668 V=800.0 PL=0
MOVL C00669 V=800.0 PL=0
MOVL C00670 V=800.0 PL=0
MOVL C00671 V=800.0 PL=0
MOVL C00672 V=800.0 PL=0
MOVL C00673 V=800.0 PL=0
MOVL C00674 V=800.0 PL=0
MOVL C00675 V=800.0 PL=0
MOVL C00676 V=800.0 PL=0
MOVL C00677 V=800.0 PL=0
MOVL C00678 V=800.0 PL=0
MOVL C00679 V=800.0 PL=0
MOVL C00680 V=800.0 PL=0
MOVL C00681 V=800.0 PL=0
MOVL C00682 V=800.0 PL=0
MOVL C00683 V=800.0 PL=0
MOVL C00684 V=800.0 PL=0
MOVL C00685 V=800.0 PL=0
MOVL C00686 V=800.0 PL=0
MOVL C00687 V=800.0 PL=0
MOVL C00688 V=800.0 PL=0
MOVL C00689 V=800.0 PL=0
MOVL C00690 V=800.0 PL=0
MOVL C00691 V=800.0 PL=0
MOVL C00692 V=800.0 PL=0
MOVL C00693 V=800.0 PL=0
MOVL C00694 V=800.0 PL=0
MOVL C00695 V=800.0 PL=0
MOVL C00696 V=800.0 PL=0
MOVL C00697 V=800.0 PL=0
MOVL C00698 V=800.0 PL=0
MOVL C00699 V=800.0 PL=0
MOVL C00700 V=800.0 PL=0
MOVL C00701 V=800.0 PL=0
MOVL C00702 V=800.0 PL=0
MOVL C00703 V=800.0 PL=0
MOVL C00704 V=800.0 PL=0
MOVL C00705 V=800.0 PL=0
MOVL C00706 V=800.0 PL=0
MOVL C00707 V=800.0 PL=0
MOVL C00708 V=800.0 PL=0
MOVL C00709 V=800.0 PL=0
MOVL C00710 V=800.0 PL=0
MOVL C00711 V=800.0 PL=0
MOVL C00712 V=800.0 PL=0
MOVL C00713 V=800.0 PL=0
MOVL C00714 V=800.0 PL=0
MOVL C00715 V=800.0 PL=0
MOVL C00716 V=800.0 PL=0
MOVL C00717 V=800.0 PL=0
MOVL C00718 V=800.0 PL=0
MOVL C00719 V=800.0 PL=0
MOVL C00720 V=800.0 PL=0
MOVL C00721 V=800.0 PL=0
MOVL C00722 V=800.0 PL=0
MOVL C00723 V=800.0 PL=0
MOVL C00724 V=800.0 PL=0
MOVL C00725 V=800.0 PL=0
MOVL C00726 V=800.0 PL=0
MOVL C00727 V=800.0 PL=0
MOVL C00728 V=800.0 PL=0
MOVL C00729 V=800.0 PL=0
MOVL C00730 V=800.0 PL=0
MOVL C00731 V=800.0 PL=0
MOVL C00732 V=800.0 PL=0
MOVL C00733 V=800.0 PL=0
MOVL C00734 V=800.0 PL=0
MOVL C00735 V=800.0 PL=0
MOVL C00736 V=800.0 PL=0
MOVL C00737 V=800.0 PL=0
MOVL C00738 V=800.0 PL=0
MOVL C00739 V=800.0 PL=0
MOVL C00740 V=800.0 PL=0
MOVL C00741 V=800.0 PL=0
MOVL C00742 V=800.0 PL=0
MOVL C00743 V=800.0 PL=0
MOVL C00744 V=800.0 PL=0
MOVL C00745 V=800.0 PL=0
MOVL C00746 V=800.0 PL=0
MOVL C00747 V=800.0 PL=0
MOVL C00748 V=800.0 PL=0
MOVL C00749 V=800.0 PL=0
MOVL C00750 V=800.0 PL=0
MOVL C00751 V=800.0 PL=0
MOVL C00752 V=800.0 PL=0
MOVL C00753 V=800.0 PL=0
MOVL C00754 V=800.0 PL=0
MOVL C00755 V=800.0 PL=0
MOVL C00756 V=800.0 PL=0
MOVL C00757 V=800.0 PL=0
MOVL C00758 V=800.0 PL=0
MOVL C00759 V=800.0 PL=0
MOVL C00760 V=800.0 PL=0
MOVL C00761 V=800.0 PL=0
MOVL C00762 V=800.0 PL=0
MOVL C00763 V=800.0 PL=0
MOVL C00764 V=800.0 PL=0
MOVL C00765 V=800.0 PL=0
MOVL C00766 V=800.0 PL=0
MOVL C00767 V=800.0 PL=0
MOVL C00768 V=800.0 PL=0
MOVL C00769 V=800.0 PL=0
MOVL C00770 V=800.0 PL=0
MOVL C00771 V=800.0 PL=0
MOVL C00772 V=800.0 PL=0
MOVL C00773 V=800.0 PL=0
MOVL C00774 V=800.0 PL=0
MOVL C00775 V=800.0 PL=0
MOVL C00776 V=800.0 PL=0
MOVL C00777 V=800.0 PL=0
MOVL C00778 V=800.0 PL=0
MOVL C00779 V=800.0 PL=0
MOVL C00780 V=800.0 PL=0
MOVL C00781 V=800.0 PL=0
MOVL C00782 V=800.0 PL=0
MOVL C00783 V=800.0 PL=0
MOVL C00784 V=800.0 PL=0
MOVL C00785 V=800.0 PL=0
MOVL C00786 V=800.0 PL=0
MOVL C00787 V=800.0 PL=0
MOVL C00788 V=800.0 PL=0
MOVL C00789 V=800.0 PL=0
MOVL C00790 V=800.0 PL=0
MOVL C00791 V=800.0 PL=0
MOVL C00792 V=800.0 PL=0
MOVL C00793 V=800.0 PL=0
MOVL C00794 V=800.0 PL=0
MOVL C00795 V=800.0 PL=0
MOVL C00796 V=800.0 PL=0
MOVL C00797 V=800.0 PL=0
MOVL C00798 V=800.0 PL=0
MOVL C00799 V=800.0 PL=0
MOVL C00800 V=800.0 PL=0
MOVL C00801 V=800.0 PL=0
MOVL C00802 V=800.0 PL=0
MOVL C00803 V=800.0 PL=0
MOVL C00804 V=800.0 PL=0
MOVL C00805 V=800.0 PL=0
MOVL C00806 V=800.0 PL=0
MOVL C00807 V=800.0 PL=0
MOVL C00808 V=800.0 PL=0
MOVL C00809 V=800.0 PL=0
MOVL C00810 V=800.0 PL=0
MOVL C00811 V=800.0 PL=0
MOVL C00812 V=800.0 PL=0
MOVL C00813 V=800.0 PL=0
MOVL C00814 V=800.0 PL=0
MOVL C00815 V=800.0 PL=0
MOVL C00816 V=800.0 PL=0
MOVL C00817 V=800.0 PL=0
MOVL C00818 V=800.0 PL=0
MOVL C00819 V=800.0 PL=0
MOVL C00820 V=800.0 PL=0
MOVL C00821 V=800.0 PL=0
MOVL C00822 V=800.0 PL=0
MOVL C00823 V=800.0 PL=0
MOVL C00824 V=800.0 PL=0
MOVL C00825 V=800.0 PL=0
MOVL C00826 V=800.0 PL=0
MOVL C00827 V=800.0 PL=0
MOVL C00828 V=800.0 PL=0
MOVL C00829 V=800.0 PL=0
MOVL C00830 V=800.0 PL=0
MOVL C00831 V=800.0 PL=0
MOVL C00832 V=800.0 PL=0
MOVL C00833 V=800.0 PL=0
MOVL C00834 V=800.0 PL=0
MOVL C00835 V=800.0 PL=0
MOVL C00836 V=800.0 PL=0
MOVL C00837 V=800.0 PL=0
MOVL C00838 V=800.0 PL=0
MOVL C00839 V=800.0 PL=0
MOVL C00840 V=800.0 PL=0
MOVL C00841 V=800.0 PL=0
MOVL C00842 V=800.0 PL=0
MOVL C00843 V=800.0 PL=0
MOVL C00844 V=800.0 PL=0
MOVL C00845 V=800.0 PL=0
MOVL C00846 V=800.0 PL=0
MOVL C00847 V=800.0 PL=0
MOVL C00848 V=800.0 PL=0
MOVL C00849 V=800.0 PL=0
MOVL C00850 V=800.0 PL=0
MOVL C00851 V=800.0 PL=0
MOVL C00852 V=800.0 PL=0
MOVL C00853 V=800.0 PL=0
MOVL C00854 V=800.0 PL=0
MOVL C00855 V=800.0 PL=0
MOVL C00856 V=800.0 PL=0
MOVL C00857 V=800.0 PL=0
MOVL C00858 V=800.0 PL=0
MOVL C00859 V=800.0 PL=0
MOVL C00860 V=800.0 PL=0
MOVL C00861 V=800.0 PL=0
MOVL C00862 V=800.0 PL=0
MOVL C00863 V=800.0 PL=0
MOVL C00864 V=800.0 PL=0
MOVL C00865 V=800.0 PL=0
MOVL C00866 V=800.0 PL=0
MOVL C00867 V=800.0 PL=0
MOVL C00868 V=800.0 PL=0
MOVL C00869 V=800.0 PL=0
MOVL C00870 V=800.0 PL=0
MOVL C00871 V=800.0 PL=0
MOVL C00872 V=800.0 PL=0
MOVL C00873 V=800.0 PL=0
MOVL C00874 V=800.0 PL=0
MOVL C00875 V=800.0 PL=0
MOVL C00876 V=800.0 PL=0
MOVL C00877 V=800.0 PL=0
MOVL C00878 V=800.0 PL=0
MOVL C00879 V=800.0 PL=0
MOVL C00880 V=800.0 PL=0
MOVL C00881 V=800.0 PL=0
MOVL C00882 V=800.0 PL=0
MOVL C00883 V=800.0 PL=0
MOVL C00884 V=800.0 PL=0
MOVL C00885 V=800.0 PL=0
MOVL C00886 V=800.0 PL=0
MOVL C00887 V=800.0 PL=0
MOVL C00888 V=800.0 PL=0
MOVL C00889 V=800.0 PL=0
MOVL C00890 V=800.0 PL=0
MOVL C00891 V=800.0 PL=0
MOVL C00892 V=800.0 PL=0
MOVL C00893 V=800.0 PL=0
MOVL C00894 V=800.0 PL=0
MOVL C00895 V=800.0 PL=0
MOVL C00896 V=800.0 PL=0
MOVL C00897 V=800.0 PL=0
MOVL C00898 V=800.0 PL=0
MOVL C00899 V=800.0 PL=0
MOVL C00900 V=800.0 PL=0
MOVL C00901 V=800.0 PL=0
MOVL C00902 V=800.0 PL=0
MOVL C00903 V=800.0 PL=0
MOVL C00904 V=800.0 PL=0
MOVL C00905 V=800.0 PL=0
MOVL C00906 V=800.0 PL=0
MOVL C00907 V=800.0 PL=0
MOVL C00908 V=800.0 PL=0
MOVL C00909 V=800.0 PL=0
MOVL C00910 V=800.0 PL=0
MOVL C00911 V=800.0 PL=0
MOVL C00912 V=800.0 PL=0
MOVL C00913 V=800.0 PL=0
MOVL C00914 V=800.0 PL=0
MOVL C00915 V=800.0 PL=0
MOVL C00916 V=800.0 PL=0
MOVL C00917 V=800.0 PL=0
MOVL C00918 V=800.0 PL=0
MOVL C00919 V=800.0 PL=0
MOVL C00920 V=800.0 PL=0
MOVL C00921 V=800.0 PL=0
MOVL C00922 V=800.0 PL=0
MOVL C00923 V=800.0 PL=0
MOVL C00924 V=800.0 PL=0
MOVL C00925 V=800.0 PL=0
MOVL C00926 V=800.0 PL=0
MOVL C00927 V=800.0 PL=0
MOVL C00928 V=800.0 PL=0
MOVL C00929 V=800.0 PL=0
MOVL C00930 V=800.0 PL=0
MOVL C00931 V=800.0 PL=0
MOVL C00932 V=800.0 PL=0
MOVL C00933 V=800.0 PL=0
MOVL C00934 V=800.0 PL=0
MOVL C00935 V=800.0 PL=0
MOVL C00936 V=800.0 PL=0
MOVL C00937 V=800.0 PL=0
MOVL C00938 V=800.0 PL=0
MOVL C00939 V=800.0 PL=0
MOVL C00940 V=800.0 PL=0
MOVL C00941 V=800.0 PL=0
MOVL C00942 V=800.0 PL=0
MOVL C00943 V=800.0 PL=0
MOVL C00944 V=800.0 PL=0
MOVL C00945 V=800.0 PL=0
MOVL C00946 V=800.0 PL=0
MOVL C00947 V=800.0 PL=0
MOVL C00948 V=800.0 PL=0
MOVL C00949 V=800.0 PL=0
MOVL C00950 V=800.0 PL=0
MOVL C00951 V=800.0 PL=0
MOVL C00952 V=800.0 PL=0
MOVL C00953 V=800.0 PL=0
MOVL C00954 V=800.0 PL=0
MOVL C00955 V=800.0 PL=0
MOVL C00956 V=800.0 PL=0
MOVL C00957 V=800.0 PL=0
MOVL C00958 V=800.0 PL=0
MOVL C00959 V=800.0 PL=0
MOVL C00960 V=800.0 PL=0
MOVL C00961 V=800.0 PL=0
MOVL C00962 V=800.0 PL=0
MOVL C00963 V=800.0 PL=0
MOVL C00964 V=800.0 PL=0
MOVL C00965 V=800.0 PL=0
MOVL C00966 V=800.0 PL=0
MOVL C00967 V=800.0 PL=0
MOVL C00968 V=800.0 PL=0
MOVL C00969 V=800.0 PL=0
MOVL C00970 V=800.0 PL=0
MOVL C00971 V=800.0 PL=0
MOVL C00972 V=800.0 PL=0
MOVL C00973 V=800.0 PL=0
MOVL C00974 V=800.0 PL=0
MOVL C00975 V=800.0 PL=0
MOVL C00976 V=800.0 PL=0
MOVL C00977 V=800.0 PL=0
MOVL C00978 V=800.0 PL=0
MOVL C00979 V=800.0 PL=0
MOVL C00980 V=800.0 PL=0
MOVL C00981 V=800.0 PL=0
MOVL C00982 V=800.0 PL=0
MOVL C00983 V=800.0 PL=0
MOVL C00984 V=800.0 PL=0
MOVL C00985 V=800.0 PL=0
MOVL C00986 V=800.0 PL=0
MOVL C00987 V=800.0 PL=0
MOVL C00988 V=800.0 PL=0
MOVL C00989 V=800.0 PL=0
MOVL C00990 V=800.0 PL=0
MOVL C00991 V=800.0 PL=0
MOVL C00992 V=800.0 PL=0
MOVL C00993 V=800.0 PL=0
MOVL C00994 V=800.0 PL=0
MOVL C00995 V=800.0 PL=0
MOVL C00996 V=800.0 PL=0
MOVL C00997 V=800.0 PL=0
MOVL C00998 V=800.0 PL=0
MOVL C00999 V=800.0 PL=0
MOVL C01000 V=800.0 PL=0
MOVL C01001 V=800.0 PL=0
MOVL C01002 V=800.0 PL=0
MOVL C01003 V=800.0 PL=0
MOVL C01004 V=800.0 PL=0
MOVL C01005 V=800.0 PL=0
MOVL C01006 V=800.0 PL=0
MOVL C01007 V=800.0 PL=0
MOVL C01008 V=800.0 PL=0
MOVL C01009 V=800.0 PL=0
MOVL C01010 V=800.0 PL=0
MOVL C01011 V=800.0 PL=0
MOVL C01012 V=800.0 PL=0
MOVL C01013 V=800.0 PL=0
MOVL C01014 V=800.0 PL=0
MOVL C01015 V=800.0 PL=0
MOVL C01016 V=800.0 PL=0
MOVL C01017 V=800.0 PL=0
MOVL C01018 V=800.0 PL=0
MOVL C01019 V=800.0 PL=0
MOVL C01020 V=800.0 PL=0
MOVL C01021 V=800.0 PL=0
MOVL C01022 V=800.0 PL=0
MOVL C01023 V=800.0 PL=0
MOVL C01024 V=800.0 PL=0
MOVL C01025 V=800.0 PL=0
MOVL C01026 V=800.0 PL=0
MOVL C01027 V=800.0 PL=0
MOVL C01028 V=800.0 PL=0
MOVL C01029 V=800.0 PL=0
MOVL C01030 V=800.0 PL=0
MOVL C01031 V=800.0 PL=0
MOVL C01032 V=800.0 PL=0
MOVL C01033 V=800.0 PL=0
MOVL C01034 V=800.0 PL=0
MOVL C01035 V=800.0 PL=0
MOVL C01036 V=800.0 PL=0
MOVL C01037 V=800.0 PL=0
MOVL C01038 V=800.0 PL=0
MOVL C01039 V=800.0 PL=0
MOVL C01040 V=800.0 PL=0
MOVL C01041 V=800.0 PL=0
MOVL C01042 V=800.0 PL=0
MOVL C01043 V=800.0 PL=0
MOVL C01044 V=800.0 PL=0
MOVL C01045 V=800.0 PL=0
MOVL C01046 V=800.0 PL=0
MOVL C01047 V=800.0 PL=0
MOVL C01048 V=800.0 PL=0
MOVL C01049 V=800.0 PL=0
MOVL C01050 V=800.0 PL=0
MOVL C01051 V=800.0 PL=0
MOVL C01052 V=800.0 PL=0
MOVL C01053 V=800.0 PL=0
MOVL C01054 V=800.0 PL=0
MOVL C01055 V=800.0 PL=0
MOVL C01056 V=800.0 PL=0
MOVL C01057 V=800.0 PL=0
MOVL C01058 V=800.0 PL=0
MOVL C01059 V=800.0 PL=0
MOVL C01060 V=800.0 PL=0
MOVL C01061 V=800.0 PL=0
MOVL C01062 V=800.0 PL=0
MOVL C01063 V=800.0 PL=0
MOVL C01064 V=800.0 PL=0
MOVL C01065 V=800.0 PL=0
MOVL C01066 V=800.0 PL=0
MOVL C01067 V=800.0 PL=0
MOVL C01068 V=800.0 PL=0
MOVL C01069 V=800.0 PL=0
MOVL C01070 V=800.0 PL=0
MOVL C01071 V=800.0 PL=0
MOVL C01072 V=800.0 PL=0
MOVL C01073 V=800.0 PL=0
MOVL C01074 V=800.0 PL=0
MOVL C01075 V=800.0 PL=0
MOVL C01076 V=800.0 PL=0
MOVL C01077 V=800.0 PL=0
MOVL C01078 V=800.0 PL=0
MOVL C01079 V=800.0 PL=0
MOVL C01080 V=800.0 PL=0
MOVL C01081 V=800.0 PL=0
MOVL C01082 V=800.0 PL=0
MOVL C01083 V=800.0 PL=0
MOVL C01084 V=800.0 PL=0
MOVL C01085 V=800.0 PL=0
MOVL C01086 V=800.0 PL=0
MOVL C01087 V=800.0 PL=0
MOVL C01088 V=800.0 PL=0
MOVL C01089 V=800.0 PL=0
MOVL C01090 V=800.0 PL=0
MOVL C01091 V=800.0 PL=0
MOVL C01092 V=800.0 PL=0
MOVL C01093 V=800.0 PL=0
MOVL C01094 V=800.0 PL=0
MOVL C01095 V=800.0 PL=0
MOVL C01096 V=800.0 PL=0
MOVL C01097 V=800.0 PL=0
MOVL C01098 V=800.0 PL=0
MOVL C01099 V=800.0 PL=0
MOVL C01100 V=800.0 PL=0
MOVL C01101 V=800.0 PL=0
MOVL C01102 V=800.0 PL=0
MOVL C01103 V=800.0 PL=0
MOVL C01104 V=800.0 PL=0
MOVL C01105 V=800.0 PL=0
MOVL C01106 V=800.0 PL=0
MOVL C01107 V=800.0 PL=0
MOVL C01108 V=800.0 PL=0
MOVL C01109 V=800.0 PL=0
MOVL C01110 V=800.0 PL=0
MOVL C01111 V=800.0 PL=0
MOVL C01112 V=800.0 PL=0
MOVL C01113 V=800.0 PL=0
MOVL C01114 V=800.0 PL=0
MOVL C01115 V=800.0 PL=0
MOVL C01116 V=800.0 PL=0
MOVL C01117 V=800.0 PL=0
MOVL C01118 V=800.0 PL=0
MOVL C01119 V=800.0 PL=0
MOVL C01120 V=800.0 PL=0
MOVL C01121 V=800.0 PL=0
MOVL C01122 V=800.0 PL=0
MOVL C01123 V=800.0 PL=0
MOVL C01124 V=800.0 PL=0
MOVL C01125 V=800.0 PL=0
MOVL C01126 V=800.0 PL=0
MOVL C01127 V=800.0 PL=0
MOVL C01128 V=800.0 PL=0
MOVL C01129 V=800.0 PL=0
MOVL C01130 V=800.0 PL=0
MOVL C01131 V=800.0 PL=0
MOVL C01132 V=800.0 PL=0
MOVL C01133 V=800.0 PL=0
MOVL C01134 V=800.0 PL=0
MOVL C01135 V=800.0 PL=0
MOVL C01136 V=800.0 PL=0
MOVL C01137 V=800.0 PL=0
MOVL C01138 V=800.0 PL=0
MOVL C01139 V=800.0 PL=0
MOVL C01140 V=800.0 PL=0
MOVL C01141 V=800.0 PL=0
MOVL C01142 V=800.0 PL=0
MOVL C01143 V=800.0 PL=0
MOVL C01144 V=800.0 PL=0
MOVL C01145 V=800.0 PL=0
MOVL C01146 V=800.0 PL=0
MOVL C01147 V=800.0 PL=0
MOVL C01148 V=800.0 PL=0
MOVL C01149 V=800.0 PL=0
MOVL C01150 V=800.0 PL=0
MOVL C01151 V=800.0 PL=0
MOVL C01152 V=800.0 PL=0
MOVL C01153 V=800.0 PL=0
MOVL C01154 V=800.0 PL=0
MOVL C01155 V=800.0 PL=0
MOVL C01156 V=800.0 PL=0
MOVL C01157 V=800.0 PL=0
MOVL C01158 V=800.0 PL=0
MOVL C01159 V=800.0 PL=0
MOVL C01160 V=800.0 PL=0
MOVL C01161 V=800.0 PL=0
MOVL C01162 V=800.0 PL=0
MOVL C01163 V=800.0 PL=0
MOVL C01164 V=800.0 PL=0
MOVL C01165 V=800.0 PL=0
MOVL C01166 V=800.0 PL=0
MOVL C01167 V=800.0 PL=0
MOVL C01168 V=800.0 PL=0
MOVL C01169 V=800.0 PL=0
MOVL C01170 V=800.0 PL=0
MOVL C01171 V=800.0 PL=0
MOVL C01172 V=800.0 PL=0
MOVL C01173 V=800.0 PL=0
MOVL C01174 V=800.0 PL=0
MOVL C01175 V=800.0 PL=0
MOVL C01176 V=800.0 PL=0
MOVL C01177 V=800.0 PL=0
MOVL C01178 V=800.0 PL=0
MOVL C01179 V=800.0 PL=0
MOVL C01180 V=800.0 PL=0
MOVL C01181 V=800.0 PL=0
MOVL C01182 V=800.0 PL=0
MOVL C01183 V=800.0 PL=0
MOVL C01184 V=800.0 PL=0
MOVL C01185 V=800.0 PL=0
MOVL C01186 V=800.0 PL=0
MOVL C01187 V=800.0 PL=0
MOVL C01188 V=800.0 PL=0
MOVL C01189 V=800.0 PL=0
MOVL C01190 V=800.0 PL=0
MOVL C01191 V=800.0 PL=0
MOVL C01192 V=800.0 PL=0
MOVL C01193 V=800.0 PL=0
MOVL C01194 V=800.0 PL=0
MOVL C01195 V=800.0 PL=0
MOVL C01196 V=800.0 PL=0
MOVL C01197 V=800.0 PL=0
MOVL C01198 V=800.0 PL=0
MOVL C01199 V=800.0 PL=0
MOVL C01200 V=800.0 PL=0
MOVL C01201 V=800.0 PL=0
MOVL C01202 V=800.0 PL=0
MOVL C01203 V=800.0 PL=0
MOVL C01204 V=800.0 PL=0
MOVL C01205 V=800.0 PL=0
MOVL C01206 V=800.0 PL=0
MOVL C01207 V=800.0 PL=0
MOVL C01208 V=800.0 PL=0
MOVL C01209 V=800.0 PL=0
MOVL C01210 V=800.0 PL=0
MOVL C01211 V=800.0 PL=0
MOVL C01212 V=800.0 PL=0
MOVL C01213 V=800.0 PL=0
MOVL C01214 V=800.0 PL=0
MOVL C01215 V=800.0 PL=0
MOVL C01216 V=800.0 PL=0
MOVL C01217 V=800.0 PL=0
MOVL C01218 V=800.0 PL=0
MOVL C01219 V=800.0 PL=0
MOVL C01220 V=800.0 PL=0
MOVL C01221 V=800.0 PL=0
MOVL C01222 V=800.0 PL=0
MOVL C01223 V=800.0 PL=0
MOVL C01224 V=800.0 PL=0
MOVL C01225 V=800.0 PL=0
MOVL C01226 V=800.0 PL=0
MOVL C01227 V=800.0 PL=0
MOVL C01228 V=800.0 PL=0
MOVL C01229 V=800.0 PL=0
MOVL C01230 V=800.0 PL=0
MOVL C01231 V=800.0 PL=0
MOVL C01232 V=800.0 PL=0
MOVL C01233 V=800.0 PL=0
MOVL C01234 V=800.0 PL=0
MOVL C01235 V=800.0 PL=0
MOVL C01236 V=800.0 PL=0
MOVL C01237 V=800.0 PL=0
MOVL C01238 V=800.0 PL=0
MOVL C01239 V=800.0 PL=0
MOVL C01240 V=800.0 PL=0
MOVL C01241 V=800.0 PL=0
MOVL C01242 V=800.0 PL=0
MOVL C01243 V=800.0 PL=0
MOVL C01244 V=800.0 PL=0
MOVL C01245 V=800.0 PL=0
MOVL C01246 V=800.0 PL=0
MOVL C01247 V=800.0 PL=0
MOVL C01248 V=800.0 PL=0
MOVL C01249 V=800.0 PL=0
MOVL C01250 V=800.0 PL=0
MOVL C01251 V=800.0 PL=0
MOVL C01252 V=800.0 PL=0
MOVL C01253 V=800.0 PL=0
MOVL C01254 V=800.0 PL=0
MOVL C01255 V=800.0 PL=0
MOVL C01256 V=800.0 PL=0
MOVL C01257 V=800.0 PL=0
MOVL C01258 V=800.0 PL=0
MOVL C01259 V=800.0 PL=0
MOVL C01260 V=800.0 PL=0
MOVL C01261 V=800.0 PL=0
MOVL C01262 V=800.0 PL=0
MOVL C01263 V=800.0 PL=0
MOVL C01264 V=800.0 PL=0
MOVL C01265 V=800.0 PL=0
MOVL C01266 V=800.0 PL=0
MOVL C01267 V=800.0 PL=0
MOVL C01268 V=800.0 PL=0
MOVL C01269 V=800.0 PL=0
MOVL C01270 V=800.0 PL=0
MOVL C01271 V=800.0 PL=0
MOVL C01272 V=800.0 PL=0
MOVL C01273 V=800.0 PL=0
MOVL C01274 V=800.0 PL=0
MOVL C01275 V=800.0 PL=0
MOVL C01276 V=800.0 PL=0
MOVL C01277 V=800.0 PL=0
MOVL C01278 V=800.0 PL=0
MOVL C01279 V=800.0 PL=0
MOVL C01280 V=800.0 PL=0
MOVL C01281 V=800.0 PL=0
MOVL C01282 V=800.0 PL=0
MOVL C01283 V=800.0 PL=0
MOVL C01284 V=800.0 PL=0
MOVL C01285 V=800.0 PL=0
MOVL C01286 V=800.0 PL=0
MOVL C01287 V=800.0 PL=0
MOVL C01288 V=800.0 PL=0
MOVL C01289 V=800.0 PL=0
MOVL C01290 V=800.0 PL=0
MOVL C01291 V=800.0 PL=0
MOVL C01292 V=800.0 PL=0
MOVL C01293 V=800.0 PL=0
MOVL C01294 V=800.0 PL=0
MOVL C01295 V=800.0 PL=0
MOVL C01296 V=800.0 PL=0
MOVL C01297 V=800.0 PL=0
MOVL C01298 V=800.0 PL=0
MOVL C01299 V=800.0 PL=0
MOVL C01300 V=800.0 PL=0
MOVL C01301 V=800.0 PL=0
MOVL C01302 V=800.0 PL=0
MOVL C01303 V=800.0 PL=0
MOVL C01304 V=800.0 PL=0
MOVL C01305 V=800.0 PL=0
MOVL C01306 V=800.0 PL=0
MOVL C01307 V=800.0 PL=0
MOVL C01308 V=800.0 PL=0
MOVL C01309 V=800.0 PL=0
MOVL C01310 V=800.0 PL=0
MOVL C01311 V=800.0 PL=0
MOVL C01312 V=800.0 PL=0
MOVL C01313 V=800.0 PL=0
MOVL C01314 V=800.0 PL=0
MOVL C01315 V=800.0 PL=0
MOVL C01316 V=800.0 PL=0
MOVL C01317 V=800.0 PL=0
MOVL C01318 V=800.0 PL=0
MOVL C01319 V=800.0 PL=0
MOVL C01320 V=800.0 PL=0
MOVL C01321 V=800.0 PL=0
MOVL C01322 V=800.0 PL=0
MOVL C01323 V=800.0 PL=0
MOVL C01324 V=800.0 PL=0
MOVL C01325 V=800.0 PL=0
MOVL C01326 V=800.0 PL=0
MOVL C01327 V=800.0 PL=0
MOVL C01328 V=800.0 PL=0
MOVL C01329 V=800.0 PL=0
MOVL C01330 V=800.0 PL=0
MOVL C01331 V=800.0 PL=0
MOVL C01332 V=800.0 PL=0
MOVL C01333 V=800.0 PL=0
MOVL C01334 V=800.0 PL=0
MOVL C01335 V=800.0 PL=0
MOVL C01336 V=800.0 PL=0
MOVL C01337 V=800.0 PL=0
MOVL C01338 V=800.0 PL=0
MOVL C01339 V=800.0 PL=0
MOVL C01340 V=800.0 PL=0
MOVL C01341 V=800.0 PL=0
MOVL C01342 V=800.0 PL=0
MOVL C01343 V=800.0 PL=0
MOVL C01344 V=800.0 PL=0
MOVL C01345 V=800.0 PL=0
MOVL C01346 V=800.0 PL=0
MOVL C01347 V=800.0 PL=0
MOVL C01348 V=800.0 PL=0
MOVL C01349 V=800.0 PL=0
MOVL C01350 V=800.0 PL=0
MOVL C01351 V=800.0 PL=0
MOVL C01352 V=800.0 PL=0
MOVL C01353 V=800.0 PL=0
MOVL C01354 V=800.0 PL=0
MOVL C01355 V=800.0 PL=0
MOVL C01356 V=800.0 PL=0
MOVL C01357 V=800.0 PL=0
MOVL C01358 V=800.0 PL=0
MOVL C01359 V=800.0 PL=0
MOVL C01360 V=800.0 PL=0
MOVL C01361 V=800.0 PL=0
MOVL C01362 V=800.0 PL=0
MOVL C01363 V=800.0 PL=0
MOVL C01364 V=800.0 PL=0
MOVL C01365 V=800.0 PL=0
MOVL C01366 V=800.0 PL=0
MOVL C01367 V=800.0 PL=0
MOVL C01368 V=800.0 PL=0
MOVL C01369 V=800.0 PL=0
MOVL C01370 V=800.0 PL=0
MOVL C01371 V=800.0 PL=0
MOVL C01372 V=800.0 PL=0
MOVL C01373 V=800.0 PL=0
MOVL C01374 V=800.0 PL=0
MOVL C01375 V=800.0 PL=0
MOVL C01376 V=800.0 PL=0
MOVL C01377 V=800.0 PL=0
MOVL C01378 V=800.0 PL=0
MOVL C01379 V=800.0 PL=0
MOVL C01380 V=800.0 PL=0
MOVL C01381 V=800.0 PL=0
MOVL C01382 V=800.0 PL=0
MOVL C01383 V=800.0 PL=0
MOVL C01384 V=800.0 PL=0
MOVL C01385 V=800.0 PL=0
MOVL C01386 V=800.0 PL=0
MOVL C01387 V=800.0 PL=0
MOVL C01388 V=800.0 PL=0
MOVL C01389 V=800.0 PL=0
MOVL C01390 V=800.0 PL=0
MOVL C01391 V=800.0 PL=0
MOVL C01392 V=800.0 PL=0
MOVL C01393 V=800.0 PL=0
MOVL C01394 V=800.0 PL=0
MOVL C01395 V=800.0 PL=0
MOVL C01396 V=800.0 PL=0
MOVL C01397 V=800.0 PL=0
MOVL C01398 V=800.0 PL=0
MOVL C01399 V=800.0 PL=0
MOVL C01400 V=800.0 PL=0
MOVL C01401 V=800.0 PL=0
MOVL C01402 V=800.0 PL=0
MOVL C01403 V=800.0 PL=0
MOVL C01404 V=800.0 PL=0
MOVL C01405 V=800.0 PL=0
MOVL C01406 V=800.0 PL=0
MOVL C01407 V=800.0 PL=0
MOVL C01408 V=800.0 PL=0
MOVL C01409 V=800.0 PL=0
MOVL C01410 V=800.0 PL=0
MOVL C01411 V=800.0 PL=0
MOVL C01412 V=800.0 PL=0
MOVL C01413 V=800.0 PL=0
MOVL C01414 V=800.0 PL=0
MOVL C01415 V=800.0 PL=0
MOVL C01416 V=800.0 PL=0
MOVL C01417 V=800.0 PL=0
MOVL C01418 V=800.0 PL=0
MOVL C01419 V=800.0 PL=0
MOVL C01420 V=800.0 PL=0
MOVL C01421 V=800.0 PL=0
MOVL C01422 V=800.0 PL=0
MOVL C01423 V=800.0 PL=0
MOVL C01424 V=800.0 PL=0
MOVL C01425 V=800.0 PL=0
MOVL C01426 V=800.0 PL=0
MOVL C01427 V=800.0 PL=0
MOVL C01428 V=800.0 PL=0
MOVL C01429 V=800.0 PL=0
MOVL C01430 V=800.0 PL=0
MOVL C01431 V=800.0 PL=0
MOVL C01432 V=800.0 PL=0
MOVL C01433 V=800.0 PL=0
MOVL C01434 V=800.0 PL=0
MOVL C01435 V=800.0 PL=0
MOVL C01436 V=800.0 PL=0
MOVL C01437 V=800.0 PL=0
MOVL C01438 V=800.0 PL=0
MOVL C01439 V=800.0 PL=0
MOVL C01440 V=800.0 PL=0
MOVL C01441 V=800.0 PL=0
MOVL C01442 V=800.0 PL=0
MOVL C01443 V=800.0 PL=0
MOVL C01444 V=800.0 PL=0
MOVL C01445 V=800.0 PL=0
MOVL C01446 V=800.0 PL=0
MOVL C01447 V=800.0 PL=0
MOVL C01448 V=800.0 PL=0
MOVL C01449 V=800.0 PL=0
MOVL C01450 V=800.0 PL=0
MOVL C01451 V=800.0 PL=0
MOVL C01452 V=800.0 PL=0
MOVL C01453 V=800.0 PL=0
MOVL C01454 V=800.0 PL=0
MOVL C01455 V=800.0 PL=0
MOVL C01456 V=800.0 PL=0
MOVL C01457 V=800.0 PL=0
MOVL C01458 V=800.0 PL=0
MOVL C01459 V=800.0 PL=0
MOVL C01460 V=800.0 PL=0
MOVL C01461 V=800.0 PL=0
MOVL C01462 V=800.0 PL=0
MOVL C01463 V=800.0 PL=0
MOVL C01464 V=800.0 PL=0
MOVL C01465 V=800.0 PL=0
MOVL C01466 V=800.0 PL=0
MOVL C01467 V=800.0 PL=0
MOVL C01468 V=800.0 PL=0
MOVL C01469 V=800.0 PL=0
MOVL C01470 V=800.0 PL=0
MOVL C01471 V=800.0 PL=0
MOVL C01472 V=800.0 PL=0
MOVL C01473 V=800.0 PL=0
MOVL C01474 V=800.0 PL=0
MOVL C01475 V=800.0 PL=0
MOVL C01476 V=800.0 PL=0
MOVL C01477 V=800.0 PL=0
MOVL C01478 V=800.0 PL=0
MOVL C01479 V=800.0 PL=0
MOVL C01480 V=800.0 PL=0
MOVL C01481 V=800.0 PL=0
MOVL C01482 V=800.0 PL=0
MOVL C01483 V=800.0 PL=0
MOVL C01484 V=800.0 PL=0
MOVL C01485 V=800.0 PL=0
MOVL C01486 V=800.0 PL=0
MOVL C01487 V=800.0 PL=0
MOVL C01488 V=800.0 PL=0
MOVL C01489 V=800.0 PL=0
MOVL C01490 V=800.0 PL=0
MOVL C01491 V=800.0 PL=0
MOVL C01492 V=800.0 PL=0
MOVL C01493 V=800.0 PL=0
MOVL C01494 V=800.0 PL=0
MOVL C01495 V=800.0 PL=0
MOVL C01496 V=800.0 PL=0
MOVL C01497 V=800.0 PL=0
MOVL C01498 V=800.0 PL=0
MOVL C01499 V=800.0 PL=0
MOVL C01500 V=800.0 PL=0
MOVL C01501 V=800.0 PL=0
MOVL C01502 V=800.0 PL=0
MOVL C01503 V=800.0 PL=0
MOVL C01504 V=800.0 PL=0
MOVL C01505 V=800.0 PL=0
MOVL C01506 V=800.0 PL=0
MOVL C01507 V=800.0 PL=0
MOVL C01508 V=800.0 PL=0
MOVL C01509 V=800.0 PL=0
MOVL C01510 V=800.0 PL=0
MOVL C01511 V=800.0 PL=0
MOVL C01512 V=800.0 PL=0
MOVL C01513 V=800.0 PL=0
MOVL C01514 V=800.0 PL=0
MOVL C01515 V=800.0 PL=0
MOVL C01516 V=800.0 PL=0
MOVL C01517 V=800.0 PL=0
MOVL C01518 V=800.0 PL=0
MOVL C01519 V=800.0 PL=0
MOVL C01520 V=800.0 PL=0
MOVL C01521 V=800.0 PL=0
MOVL C01522 V=800.0 PL=0
MOVL C01523 V=800.0 PL=0
MOVL C01524 V=800.0 PL=0
MOVL C01525 V=800.0 PL=0
MOVL C01526 V=800.0 PL=0
MOVL C01527 V=800.0 PL=0
MOVL C01528 V=800.0 PL=0
MOVL C01529 V=800.0 PL=0
MOVL C01530 V=800.0 PL=0
MOVL C01531 V=800.0 PL=0
MOVL C01532 V=800.0 PL=0
MOVL C01533 V=800.0 PL=0
MOVL C01534 V=800.0 PL=0
MOVL C01535 V=800.0 PL=0
MOVL C01536 V=800.0 PL=0
MOVL C01537 V=800.0 PL=0
MOVL C01538 V=800.0 PL=0
MOVL C01539 V=800.0 PL=0
MOVL C01540 V=800.0 PL=0
MOVL C01541 V=800.0 PL=0
MOVL C01542 V=800.0 PL=0
MOVL C01543 V=800.0 PL=0
MOVL C01544 V=800.0 PL=0
MOVL C01545 V=800.0 PL=0
MOVL C01546 V=800.0 PL=0
MOVL C01547 V=800.0 PL=0
MOVL C01548 V=800.0 PL=0
MOVL C01549 V=800.0 PL=0
MOVL C01550 V=800.0 PL=0
MOVL C01551 V=800.0 PL=0
MOVL C01552 V=800.0 PL=0
MOVL C01553 V=800.0 PL=0
MOVL C01554 V=800.0 PL=0
MOVL C01555 V=800.0 PL=0
MOVL C01556 V=800.0 PL=0
MOVL C01557 V=800.0 PL=0
MOVL C01558 V=800.0 PL=0
MOVL C01559 V=800.0 PL=0
MOVL C01560 V=800.0 PL=0
MOVL C01561 V=800.0 PL=0
MOVL C01562 V=800.0 PL=0
MOVL C01563 V=800.0 PL=0
MOVL C01564 V=800.0 PL=0
MOVL C01565 V=800.0 PL=0
MOVL C01566 V=800.0 PL=0
MOVL C01567 V=800.0 PL=0
MOVL C01568 V=800.0 PL=0
MOVL C01569 V=800.0 PL=0
MOVL C01570 V=800.0 PL=0
MOVL C01571 V=800.0 PL=0
MOVL C01572 V=800.0 PL=0
MOVL C01573 V=800.0 PL=0
MOVL C01574 V=800.0 PL=0
MOVL C01575 V=800.0 PL=0
MOVL C01576 V=800.0 PL=0
MOVL C01577 V=800.0 PL=0
MOVL C01578 V=800.0 PL=0
MOVL C01579 V=800.0 PL=0
MOVL C01580 V=800.0 PL=0
MOVL C01581 V=800.0 PL=0
MOVL C01582 V=800.0 PL=0
MOVL C01583 V=800.0 PL=0
MOVL C01584 V=800.0 PL=0
MOVL C01585 V=800.0 PL=0
MOVL C01586 V=800.0 PL=0
MOVL C01587 V=800.0 PL=0
MOVL C01588 V=800.0 PL=0
MOVL C01589 V=800.0 PL=0
MOVL C01590 V=800.0 PL=0
MOVL C01591 V=800.0 PL=0
MOVL C01592 V=800.0 PL=0
MOVL C01593 V=800.0 PL=0
MOVL C01594 V=800.0 PL=0
MOVL C01595 V=800.0 PL=0
MOVL C01596 V=800.0 PL=0
MOVL C01597 V=800.0 PL=0
MOVL C01598 V=800.0 PL=0
MOVL C01599 V=800.0 PL=0
MOVL C01600 V=800.0 PL=0
MOVL C01601 V=800.0 PL=0
MOVL C01602 V=800.0 PL=0
MOVL C01603 V=800.0 PL=0
MOVL C01604 V=800.0 PL=0
MOVL C01605 V=800.0 PL=0
MOVL C01606 V=800.0 PL=0
MOVL C01607 V=800.0 PL=0
MOVL C01608 V=800.0 PL=0
MOVL C01609 V=800.0 PL=0
MOVL C01610 V=800.0 PL=0
MOVL C01611 V=800.0 PL=0
MOVL C01612 V=800.0 PL=0
MOVL C01613 V=800.0 PL=0
MOVL C01614 V=800.0 PL=0
MOVL C01615 V=800.0 PL=0
MOVL C01616 V=800.0 PL=0
MOVL C01617 V=800.0 PL=0
MOVL C01618 V=800.0 PL=0
MOVL C01619 V=800.0 PL=0
MOVL C01620 V=800.0 PL=0
MOVL C01621 V=800.0 PL=0
MOVL C01622 V=800.0 PL=0
MOVL C01623 V=800.0 PL=0
MOVL C01624 V=800.0 PL=0
MOVL C01625 V=800.0 PL=0
MOVL C01626 V=800.0 PL=0
MOVL C01627 V=800.0 PL=0
MOVL C01628 V=800.0 PL=0
MOVL C01629 V=800.0 PL=0
MOVL C01630 V=800.0 PL=0
MOVL C01631 V=800.0 PL=0
MOVL C01632 V=800.0 PL=0
